// TwinCAT 3 PLC project Supervisorio
// ProgramVersion: 3.1.4024.0
// libraries:
//   CmpBitmapPool, * (System)
//   Tc2_Database, * (Beckhoff Automation GmbH)
//   Tc2_Standard, * (Beckhoff Automation GmbH)
//   Tc2_System, * (Beckhoff Automation GmbH)
//   Tc2_Utilities, * (Beckhoff Automation GmbH)
//   Tc3_EventLogger, * (Beckhoff Automation GmbH)
//   Tc3_Module, * (Beckhoff Automation GmbH)
//   VisuDialogs, * (System)
//   VisuSymbols,3.5.10.0,System
// project tree:
//   DUTs/ paPositions.TcDUT, raPositions.TcDUT, selectHist.TcDUT, statusEstufa.TcDUT, st_csv.TcDUT, tempData.TcDUT, timeDry.TcDUT (not stored)
//   / GlobalTextList.TcGTLO, PlcTask.TcTTO (not stored), Visualization Manager.TcVMO (not stored), VISU_TASK.TcTTO
//   GVLs/ GVL.TcGVL, GVL_C.TcGVL, GVL_P.TcGVL
//   POUs/Botons/ confirmSetInicio.TcPOU, confirmSecagem.TcPOU, gravarConfigPosicao.TcPOU, gravarConfigPosicao020.TcPOU, gravarConfigPosicao021.TcPOU, gravarConfigPosicao_Reator.TcPOU, gravarConfigPosicao_Reator_3.TcPOU, gravarConfigPosicao_Reator_2.TcPOU, iniciaProgramacaoEstufa.TcPOU, posCarrinho.TcPOU, posCarrinho2.TcPOU (not stored), posCarrinho3.TcPOU, selectPos021.TcPOU (not stored), selectPos019.TcPOU (not stored), selectPos020.TcPOU (not stored), simIniciaProg.TcPOU (not stored), simIniciaProg_Manual.TcPOU, simIniciaProg_Manual_3.TcPOU, simIniciaProg_Manual_2.TcPOU
//   POUs/ Chart_Gen.TcPOU, historical.TcPOU, MAIN.TcPOU, POU_Persistent.TcPOU, P_TextModeWrite.TcPOU, registerProc.TcPOU, registerProc20.TcPOU, registerProc21.TcPOU, registradorLog.TcPOU, registradorLog20.TcPOU, registradorLog21.TcPOU, ReportGenerator.TcPOU, Rotina019.TcPOU, Rotina019_Manual.TcPOU, Rotina021_Manual.TcPOU, Rotina020.TcPOU, Rotina021.TcPOU, Rotina020_Manual.TcPOU
//   VISUs/ Aba_Estufa.TcVIS, Aba_Estufa_2.TcVIS, Aba_Estufa_3.TcVIS (not stored), Aba_Manu.TcVIS, addComment.TcVIS, Carrinho_3.TcVIS (not stored), Carrinho_2.TcVIS (not stored), ConfigPosicao_3.TcVIS, ConfigPosicao_2.TcVIS, ConfigPosicao_Reator.TcVIS, ConfigPosicao_Reator_3.TcVIS (not stored), ConfigPosicao_Reator_2.TcVIS, Estufa2.TcVIS, Estufa3.TcVIS, FinalizaProg.TcVIS, Grafico_3.TcVIS, Grafico_2.TcVIS, Historical.TcVIS, IniciaProg_3.TcVIS, IniciaProg_2.TcVIS, Manu021.TcVIS, Manu020.TcVIS, Notifica24horas.TcVIS, Manu019.TcVIS, Carrinho.TcVIS, Estufa1.TcVIS, Grafico.TcVIS, Home.TcVIS, ImagePool.TcIPO (not stored), ConfigPosicao.TcVIS, IniciaProg.TcVIS (not stored), setInicio.TcVIS, setSecagem.TcVIS, TimeCustom.TcVIS, TimeCustom_3.TcVIS, TimeCustom_2.TcVIS
// real-time tasks:
//   TASK PlcTask: cycle T#10ms, priority 20, ADS port 350
//   TASK VISU_TASK: cycle T#200000us, priority 30, ADS port 351
// I/O:
//   DEVICE Device 1 (EtherCAT), AmsNetId 5.148.119.239.2.1
//     Term 1 (EK1200) [EK1200-5000 EtherCAT Power supply (2A E-Bus)]
//       Term 2 (EL6070) [EL6070 1Ch. Licensing-Terminal]
//       Term 3 (EL3058) [EL3058 8Ch. Ana. Input 4-20mA]
//       Term 4 (EL3052) [EL3052 2Ch. Ana. Input 4-20mA]
//       Term 5 (EL4008) [EL4008 8Ch. Ana. Output 0-10V, 12bit]
//       Term 6 (EL4002) [EL4002 2Ch. Ana. Output 0-10V, 12bit]
//       Term 7 (EL1809) [EL1809 16Ch. Dig. Input 24V, 3ms]
//       Term 8 (EL1809) [EL1809 16Ch. Dig. Input 24V, 3ms]
//       Term 9 (EL1809) [EL1809 16Ch. Dig. Input 24V, 3ms]
//       Term 10 (EL2809) [EL2809 16Ch. Dig. Output 24V, 0.5A]
//       Term 11 (EL2809) [EL2809 16Ch. Dig. Output 24V, 0.5A]
//       Term 12 (EL9011) [EL9011 End Terminal]
//   DEVICE Device 3 (NOV-DP-RAM)
// variable links:
//   Supervisorio/Supervisorio Instance <-> Device 1 (EtherCAT)/Term 1 (EK1200)/Term 10 (EL2809)
//     PlcTask Outputs/GVL.DigitalOut1[{1..16}] <-> Channel {1..16}/Output  (16 links)
//   Supervisorio/Supervisorio Instance <-> Device 1 (EtherCAT)/Term 1 (EK1200)/Term 11 (EL2809)
//     PlcTask Outputs/GVL.DigitalOut2[{1..16}] <-> Channel {1..16}/Output  (16 links)
//   Supervisorio/Supervisorio Instance <-> Device 1 (EtherCAT)/Term 1 (EK1200)/Term 3 (EL3058)
//     PlcTask Inputs/GVL.AnalogIn_4_20[{0..7}] <-> AI Standard Channel {1..8}/Value  (8 links)
//   Supervisorio/Supervisorio Instance <-> Device 1 (EtherCAT)/Term 1 (EK1200)/Term 4 (EL3052)
//     PlcTask Inputs/GVL.AnalogIn_4_20[8] <-> AI Standard Channel 1/Value
//     PlcTask Inputs/GVL.AnalogIn_4_20[9] <-> AI Standard Channel 2/Value
//   Supervisorio/Supervisorio Instance <-> Device 1 (EtherCAT)/Term 1 (EK1200)/Term 5 (EL4008)
//     PlcTask Outputs/GVL.AnalogOut_0_10[{0..7}] <-> AO Outputs Channel {1..8}/Analog output  (8 links)
//   Supervisorio/Supervisorio Instance <-> Device 1 (EtherCAT)/Term 1 (EK1200)/Term 6 (EL4002)
//     PlcTask Outputs/GVL.AnalogOut_0_10[8] <-> AO Outputs Channel 1/Analog output
//     PlcTask Outputs/GVL.AnalogOut_0_10[9] <-> AO Outputs Channel 2/Analog output
//   Supervisorio/Supervisorio Instance <-> Device 1 (EtherCAT)/Term 1 (EK1200)/Term 7 (EL1809)
//     PlcTask Inputs/GVL.DigitalIn1[{1..16}] <-> Channel {1..16}/Input  (16 links)
//   Supervisorio/Supervisorio Instance <-> Device 1 (EtherCAT)/Term 1 (EK1200)/Term 8 (EL1809)
//     PlcTask Inputs/GVL.DigitalIn2[{1..16}] <-> Channel {1..16}/Input  (16 links)
//   Supervisorio/Supervisorio Instance <-> Device 1 (EtherCAT)/Term 1 (EK1200)/Term 9 (EL1809)
//     PlcTask Inputs/GVL.DigitalIn3[{1..16}] <-> Channel {1..16}/Input  (16 links)

CONFIGURATION Supervisorio
    RESOURCE PLC ON TwinCAT3
        TASK VISU_TASK(INTERVAL := T#200000us, PRIORITY := 30);
        PROGRAM VisuElems_Visu_Prg WITH VISU_TASK : VisuElems.Visu_Prg;
    END_RESOURCE
END_CONFIGURATION

// ---- DUTs/paPositions.TcDUT
TYPE paPositions :
STRUCT
	cor: INT;
	color: DWORD;
	numOF: STRING;
	lote: STRING;
	text: string;
	class: REAL;
	pot: REAL;
	FP: INT;
	isolamento: int;
	reator: BOOL:= TRUE;
END_STRUCT
END_TYPE

// ---- DUTs/raPositions.TcDUT
TYPE raPositions :
STRUCT
	cor: INT;
	color: DWORD;
END_STRUCT
END_TYPE

// ---- DUTs/selectHist.TcDUT
TYPE selectHist :
STRUCT
	data: STRING(10);
	hora: STRING(10);
	auto: STRING(10);
	pos:  STRING(10);
	orfb: STRING(10);
	lote: STRING(10);
	class: STRING(50);
	pot: LREAL(8);
	isola: LREAL(8);
	fPot: STRING(10);
	reator: STRING(10);
	tempo: STRING(10);
	temp: DINT;
END_STRUCT
END_TYPE

// ---- DUTs/statusEstufa.TcDUT
TYPE statusEstufa :
STRUCT
	tempoSecagem: TIME; //DEFINIDO NA TELA ConfigPosicao
	tempoArmazenagem: TIME; //DEFINIDO NA TELA ConfigPosicao
	inicioSecagem: DATE_AND_TIME;
	fimSecagem: DATE_AND_TIME;
	prevFimSeca: DATE_AND_TIME;
	fimArmazenagem: DATE_AND_TIME;
	statusInicioSecagem: STRING;
	statusFimSecagem: STRING;
	statusFimArmazenagem: STRING;
	anoSec: STRING;
	mesSec: STRING;
	diaSec: STRING;
	horaSec: STRING;
	minutoSec: STRING;
	anoArm: STRING;
	mesArm: STRING;
	diaArm: STRING;
	horaArm: STRING;
	minutoArm: STRING;
	inicioReator: STRING;
	dtInicioReator: DATE_AND_TIME;
	start: BOOL;
	startManual: BOOL;
	tempSeca: INT;
	tempArm: int;
END_STRUCT
END_TYPE

// ---- DUTs/st_csv.TcDUT
TYPE st_csv :
STRUCT
	dia: STRING;
	mes: STRING;
	ano: STRING;
	ordem: STRING;
	lote: string;
END_STRUCT
END_TYPE

// ---- DUTs/tempData.TcDUT
TYPE tempData : 
STRUCT
	temp: REAL;
END_STRUCT
END_TYPE

// ---- GVLs/GVL.TcGVL
{attribute 'qualified_only'}
VAR_GLOBAL
	
////// Layout Interativo ////////

	
	
	corPos: DWORD;
	
  (*Pos Com Reator 00C000
	Pos Sem Reator FFFF00
	Pos Livre FFFFFF*)
	n: INT;
	i: INT;
	
	cfgPos_OF019: STRING;
	cfgPos_OF020: STRING;
	cfgPos_OF021: STRING;
	cfgPos_LT019: STRING;
	cfgPos_LT020: STRING;
	cfgPos_LT021: STRING;
	cfgPos_Class019: REAL;
	cfgPos_Class020: REAL;
	cfgPos_Class021: REAL;
	cfgPos_Pot019: REAL;
	cfgPos_Pot020: REAL;
	cfgPos_Pot021: REAL;
	cfgPos_Reat019: BOOL;
	cfgPos_Reat020: BOOL;
	cfgPos_Reat021: BOOL;
	cfgPos_FP019: INT;
	cfgPos_FP020: INT;
	cfgPos_FP021: INT;
	cfgPos_Iso019: INT;
	cfgPos_Iso020: INT;
	cfgPos_Iso021: INT;
	
	
	
////// Status Programação ///////////	

	
	logRegister: ARRAY[0..2] OF STRING;
	logRegister19: STRING;
	logRegister20: STRING;
	logRegister21: STRING;
	addTextLog: STRING;
	totalPos: ARRAY[0..2] OF INT;
	totalSeca: ARRAY[0..2] OF STRING;
	totalArm: ARRAY[0..2] OF STRING;
	totalRaet: ARRAY[0..2] OF INT;
	totalManual: ARRAY[0..2] OF INT;
	
	progInicio: ARRAY[0..2] OF STRING; //'DT#2024-3-31-23:59:0'
	progInicioReat: STRING;
	ano: STRING;
	mes: STRING;
	dia: STRING;
	hora: STRING;
	minuto: STRING;
	
	horaSecagem: STRING;
	minSecagem: STRING;
	horaArmazem: STRING;
	minArmazem: STRING;
	
	
	
	endSeca19: TIME;
	endSeca20: TIME;
	endSeca21: TIME;
	
	endArm19: TIME;
	endArm20: TIME;
	endArm21: TIME;
	
	
	
////// System Time ///////////	
	
	fbGetLocalSystemTime: FB_LocalSystemTime;
	sSystemDateTime: STRING;
	sSystemTime: STRING;
	sSystemDate: STRING;
	sDateTime: STRING;
	
	somaTempo: DATE_AND_TIME;
	
////// NÃO DEFINIDAS //////	
	actPos: INT;
	actEst: INT;
	actReat: INT;
	estAtiva: STRING;
	
	logButton: bool;
	
	bVentOn: BOOL;
	bAquecOn: BOOL;
	
	envialog: string;
	
	bstartchart019: BOOL;
	bstartchart020: BOOL;
	bstartchart021: BOOL;
	bAgendaInicio: BOOL;
	emergency: bool;
	
////// DECLARAÇÃO IOs //////

	AnalogIn_4_20 AT %I* : ARRAY[0..9] OF INT;
	AnalogOut_0_10 AT %Q* : ARRAY[0..9] OF INT;
	DigitalIn1 AT %I* : ARRAY[1..16] OF BOOL;
	DigitalIn2 AT %I* : ARRAY[1..16] OF BOOL;
	DigitalIn3 AT %I* : ARRAY[1..16] OF BOOL;
	DigitalOut1 AT %Q* : ARRAY[1..16] OF BOOL;
	DigitalOut2 AT %Q* : ARRAY[1..16] OF BOOL;
	
	
////// VARIAVEIS ESTUFA 019 //////

	zona1atual_019: REAL;
	zona2atual_019: REAL;
	zonaSegAtual_019: REAL;
	
	
	sobrecarga_M1_vent_019: BOOL;
	sobrecarga_M2_vent_019: BOOL;
	sobrecarga_Purga_019: BOOL;
	falhaTempHigh_019: BOOL;
	queimador1_block_019: BOOL;
	queimador2_block_019: BOOL;
	ventilacao_Ligada_019: BOOL;
	aquecimento_Desligado_019: BOOL;
	aquecimento_Ligado_019: BOOL;
	fimCicloAquecimento_019: BOOL;
	purgandoCamara_019: BOOL;
	liga_ventilacao_019: BOOL;
	liga_aquecimento_019: BOOL;
	desl_aquecimento_019: BOOL;
	emergencia019: BOOL;
	inEmergencia019: BOOL;
	
////// VARIAVEIS ESTUFA 020 //////

	zona1atual_020: REAL;
	zona2atual_020: REAL;
	zonaSegAtual_020: REAL;
	
	
	sobrecarga_M1_vent_020: BOOL;
	sobrecarga_M2_vent_020: BOOL;
	sobrecarga_Purga_020: BOOL;
	falhaTempHigh_020: BOOL;
	queimador1_block_020: BOOL;
	queimador2_block_020: BOOL;
	ventilacao_Ligada_020: BOOL;
	aquecimento_Desligado_020: BOOL;
	aquecimento_Ligado_020: BOOL;
	fimCicloAquecimento_020: BOOL;
	purgandoCamara_020: BOOL;
	liga_ventilacao_020: BOOL;
	liga_aquecimento_020: BOOL;
	desl_aquecimento_020: BOOL;	
	emergencia020: BOOL;
	inEmergencia020: BOOL;
	
////// VARIAVEIS ESTUFA 021 //////

	zona1atual_021: REAL;
	zona2atual_021: REAL;
	zonaSegAtual_021: REAL;
	
	
	sobrecarga_M1_vent_021: BOOL;
	sobrecarga_M2_vent_021: BOOL;
	sobrecarga_Purga_021: BOOL;
	falhaTempHigh_021: BOOL;
	queimador1_block_021: BOOL;
	queimador2_block_021: BOOL;
	ventilacao_Ligada_021: BOOL;
	aquecimento_Desligado_021: BOOL;
	aquecimento_Ligado_021: BOOL;
	fimCicloAquecimento_021: BOOL;
	purgandoCamara_021: BOOL;
	liga_ventilacao_021: BOOL;
	liga_aquecimento_021: BOOL;
	desl_aquecimento_021: BOOL;	
	emergencia021: BOOL;
	inEmergencia021: BOOL;
	
////// VARIAVEIS PRODWIN /////

	pwProd_019: BOOL;
	pwProd_020: BOOL;
	pwProd_021: BOOL;
	pwEmerg_019: BOOL;
	pwEmerg_020: BOOL;
	pwEmerg_021: BOOL;
	
////// VARIAVEI SQL //////

	sCmdInsertLog: STRING(3000);//INSERT INTO [dbo].[LogGeneral] ([HistoricalTime],[Description])VALUES('historicaltime','Description')
	//SELECT * FROM [dbo].[LogGeneral]
	sCmdInsertProc: STRING(3000);//INSERT INTO [dbo].[ProcessTable] ([data],[hora],[estufa],[auto],[user],[codPeca],[OF],[lote],[class],[pot],[isola],[fPot],[reator],[TIME],[temp])
	//VALUES ('data', 'hora', estufa0, 'auto', 'user', 'codpeca', 'OF', 'lote',	class0,	pot0, isola0, Fp0.0, 'reator', 'tempo',	tempe0)

	sCmdSelect19: STRING(3000);//'SELECT [data],[hora],[auto],[pos],[OF],[lote],[class],[pot],[isola],[fPot],[reator],[time],[temp] FROM [dbo].[ProcessTable19] WHERE data=$'2024-10-24$';';
	sCmdSelect20: STRING(3000);
	sCmdSelect21: STRING(3000);
	
	bInsertLog: BOOL;
	bInsertProc: BOOL;
	bSelect19: BOOL;
	aSelect19: ARRAY[1..MAX_CSV_ROWS] OF selecthist;
	bSelect20: BOOL;
	aSelect20: ARRAY[1..MAX_CSV_ROWS] OF selecthist;
	bSelect21: BOOL;
	aSelect21: ARRAY[1..MAX_CSV_ROWS] OF selecthist;
	
	permanencia: ARRAY[1..3] OF TIME;
	sReator: STRING;
	sFp: STRING;
	sIso: STRING;
	sAuto: STRING;
	bHistory: bool;
	
////// VARIAVEIS CSV //////
	
	report19: BOOL;
	radioFiltro: INT;
	radioEstufa: INT;
	radioData: BOOL;
	radioOF: BOOL;
	radioLote: BOOL;
	arrCVSfilter: ARRAY[0..2] OF st_csv;
	
	database: ARRAY[0..MAX_CSV_ROWS, 0..MAX_CSV_COLUMNS] OF STRING(MAX_CSV_FIELD_LENGTH); (*[ (* Source PLC database *)
	'0_0', '0_1', '0_2', '0_3', '0_4', '0_5',
	'1', '1_1', '1_2', '1_3', '1_4', '1_5',
	'2_0', '2_1', '2_2', '2_3', '2_4', '2_5',
	'3_0', '3_1', '3_2', '3_3', '3_4', '3_5',
	'4_0', '4_1', '4_2', '4_3', '4_4', '4_5',
	'5_0', '5_1', '5_2', '5_3', '5_4', '5_5'];*)
	
END_VAR

// ---- GVLs/GVL_C.TcGVL
VAR_GLOBAL CONSTANT
	MAX_CSV_ROWS 			: UDINT := 10000;
	MAX_CSV_COLUMNS 		: UDINT := 14;
	MAX_CSV_FIELD_LENGTH	: UDINT := 50;
END_VAR

// ---- GVLs/GVL_P.TcGVL
{attribute 'qualified_only'}
VAR_GLOBAL PERSISTENT
	
////// VARIAVEIS ESTUFA 019 //////

	zona1setpt_019: INT;
	zona2setpt_019: INT;
	zonaSegSetpt_019: INT;
	setPoint_019: INT;
	arr_Iso_1: ARRAY[0..3] OF INT;
	arr_FP_1: ARRAY[0..3] OF STRING;
	arr_CustomTime: ARRAY[0..1,1..10] OF INT;
	
////// VARIAVEIS ESTUFA 020 //////

	zona1setpt_020: INT;
	zona2setpt_020: INT;
	zonaSegSetpt_020: INT;
	setPoint_020: INT;
	arr_Iso_2: ARRAY[0..3] OF INT;
	arr_FP_2: ARRAY[0..3] OF STRING;
	arr_CustomTime_020: ARRAY[0..1,1..10] OF INT;
	
////// VARIAVEIS ESTUFA 021 //////

	zona1setpt_021: INT;
	zona2setpt_021: INT;
	zonaSegSetpt_021: INT;
	setPoint_021: INT;	
	arr_Iso_3: ARRAY[0..3] OF INT;
	arr_FP_3: ARRAY[0..3] OF STRING;
	arr_CustomTime_021: ARRAY[0..1,1..10] OF INT;
	
////// STATUS PROGRAMAÇÃO /////

	arrStatusEstufas: ARRAY[0..2] OF statusEstufa;
	etapa_process: ARRAY[0..2] OF STRING;
	
	arrLogEstufa19: ARRAY[1..100] OF STRING;
	arrLogEstufa20: ARRAY[1..100] OF STRING;
	arrLogEstufa21: ARRAY[1..100] OF STRING;
	
	
////// GRAFICO /////////

	arrTemp019: ARRAY[1..720] OF REAL;
	arrTempVisu019: ARRAY[1..720] OF REAL;
	arrTemp020: ARRAY[1..720] OF REAL;
	arrTempVisu020: ARRAY[1..720] OF REAL;
	arrTemp021: ARRAY[1..720] OF REAL;
	arrTempVisu021: ARRAY[1..720] OF REAL;
	
///// LAYOUT INTERATIVO /////

 	aReatorE019: ARRAY[1..2, 1..3] OF INT;
	aPositionsE019: ARRAY[1..24] OF paPositions;
	aReatorE020: ARRAY[1..2, 1..3] OF INT;
	aPositionsE020: ARRAY[1..24] OF paPositions;
	aReatorE021: ARRAY[1..2, 1..3] OF INT;
	aPositionsE021: ARRAY[1..24] OF paPositions;
	
	bCarrinhoReator1: BOOL:= TRUE;
	bCarrinhoReator2: BOOL:= TRUE;
	bCarrinhoReator3: BOOL:= TRUE;
	
	corPosReator1: ARRAY[1..6] OF raPositions;
	corPosReator2: ARRAY[1..6] OF raPositions;
	corPosReator3: ARRAY[1..6] OF raPositions;
	
END_VAR

// ---- POUs/Botons/confirmSetInicio.TcPOU
PROGRAM confirmSetInicio
VAR
END_VAR

gvl.progInicio[gvl.actEst]:= 'DT#20';
gvl.progInicio[gvl.actEst]:= concat(gvl.progInicio[gvl.actEst],gvl.ano);
gvl.progInicio[gvl.actEst]:= concat(gvl.progInicio[gvl.actEst],'-');
gvl.progInicio[gvl.actEst]:= concat(gvl.progInicio[gvl.actEst],gvl.mes);
gvl.progInicio[gvl.actEst]:= concat(gvl.progInicio[gvl.actEst],'-');
gvl.progInicio[gvl.actEst]:= concat(gvl.progInicio[gvl.actEst],gvl.dia);
gvl.progInicio[gvl.actEst]:= concat(gvl.progInicio[gvl.actEst],'-');
gvl.progInicio[gvl.actEst]:= concat(gvl.progInicio[gvl.actEst],gvl.hora);
gvl.progInicio[gvl.actEst]:= concat(gvl.progInicio[gvl.actEst],':');
gvl.progInicio[gvl.actEst]:= concat(gvl.progInicio[gvl.actEst],gvl.minuto);
gvl.progInicio[gvl.actEst]:= concat(gvl.progInicio[gvl.actEst],':0');

END_PROGRAM

// ---- POUs/Botons/confirmSecagem.TcPOU
PROGRAM confirmSecagem
VAR
	tempSeca: STRING;
	
END_VAR

//ESTE PROGRAMA TRANSFORMA O INPUT DO DIALOG EM TEMPO DE SECAGEM

tempSeca:= 'T#';
tempSeca:= concat(tempseca, TIME_TO_STRING(gvl_p.arrStatusEstufas[2].tempoSecagem));
tempSeca:= concat(tempseca, 'H');

GVL_p.arrStatusEstufas[2].tempoSecagem := STRING_TO_TIME(tempSeca);

END_PROGRAM

// ---- POUs/Botons/gravarConfigPosicao.TcPOU
PROGRAM gravarConfigPosicao
VAR
	bReator: ARRAY[0..2] OF BOOL;
	posicaoAtual: STRING;
	enviaLog: STRING;
	estufaAtual: STRING;
END_VAR

// CONTABILIZA A POSIÇÃO TOTAL  MUST BE FIRST-----------------------------------------------------------------

IF gvl_p.aPositionsE019[gvl.actPos].cor = 0 THEN
	gvl.totalPos[0]:= gvl.totalPos[0]+1;			
END_IF

// VERIFICA SE HA REATOR E MUDA A COR DO QUADRADO ------------------------------------
IF bReator[0] THEN
	gvl_p.aPositionsE019[gvl.actPos].cor:= 1;
	//gvl_p.bCarrinhoReator1:=TRUE;
	gvl.cfgPos_Reat019:=TRUE;
	ELSE
		gvl_p.aPositionsE019[gvl.actPos].cor:=2;
		//gvl_p.bCarrinhoReator1:=FALSE;
		gvl.cfgPos_Reat019:=FALSE;
END_IF

// REGISTRA AS INFORMAÇÕES EM CADA POSIÇÃO -------------------------------------------------------------
FOR gvl.n:=1 TO 24 BY 1 DO
	IF gvl.actPos = gvl.n THEN
		gvl_p.aPositionsE019[gvl.n].numOF:= gvl.cfgPos_OF019;
		gvl_p.aPositionsE019[gvl.n].lote:= gvl.cfgPos_LT019;
		gvl_p.aPositionsE019[gvl.n].class:= gvl.cfgPos_Class019;
		gvl_p.aPositionsE019[gvl.n].pot:= gvl.cfgPos_Pot019;
		gvl_p.aPositionsE019[gvl.n].reator:= gvl.cfgPos_Reat019;
		gvl_p.aPositionsE019[gvl.n].FP:= gvl.cfgPos_FP019;
		gvl_p.aPositionsE019[gvl.n].isolamento:= gvl.cfgPos_Iso019;
		gvl_p.aPositionsE019[gvl.n].text:= insert(gvl.cfgPos_OF019,'-',5);
		gvl_p.aPositionsE019[gvl.n].text:= concat(gvl_p.aPositionsE019[gvl.n].text,gvl.cfgPos_LT019);
	END_IF
END_FOR

// DEFINIÇÃO DOS TEMPOS DE ACORDO COM AS CLASSES ----------------------------------------------
(*IF gvl_p.aPositionsE019[gvl.actPos].class <= 15 THEN
		GVL_p.arrStatusEstufas[gvl.actEst].tempoSecagem := T#60H;
		GVL_p.arrStatusEstufas[gvl.actEst].tempoArmazenagem := T#192H;
		gvl.totalSeca[0]:= '60';
		gvl_p.arrStatusEstufas[gvl.actEst].tempSeca:= 120;
		gvl.totalArm[0]:= '192';
		gvl_p.arrStatusEstufas[gvl.actEst].tempArm:= 70;
		ELSIF gvl_p.aPositionsE019[gvl.actPos].class > 15 THEN
			GVL_p.arrStatusEstufas[gvl.actEst].tempoSecagem:= T#96H;
			GVL_p.arrStatusEstufas[gvl.actEst].tempoArmazenagem:= T#240H;
			gvl.totalSeca[0]:= '96';
			gvl_p.arrStatusEstufas[gvl.actEst].tempSeca:= 120;
			gvl.totalArm[0]:= '240';
			gvl_p.arrStatusEstufas[gvl.actEst].tempArm:= 70;
END_IF*)
IF gvl_p.aPositionsE019[gvl.actPos].pot <= 750 AND gvl_p.aPositionsE019[gvl.actPos].isolamento <= 25 AND gvl_p.aPositionsE019[gvl.actPos].FP = 1 THEN
	GVL_p.arrStatusEstufas[0].tempoSecagem := T#60H;
	GVL_p.arrStatusEstufas[0].tempoArmazenagem := T#192H;
	gvl.totalSeca[0]:= '60';
	gvl_p.arrStatusEstufas[0].tempSeca:= 120;
	gvl.totalArm[0]:= '192';
	gvl_p.arrStatusEstufas[0].tempArm:= 70;
	ELSIF gvl_p.aPositionsE019[gvl.actPos].pot <= 750 AND gvl_p.aPositionsE019[gvl.actPos].isolamento > 25 AND gvl_p.aPositionsE019[gvl.actPos].FP = 1 THEN
		GVL_p.arrStatusEstufas[0].tempoSecagem:= T#96H;
		GVL_p.arrStatusEstufas[0].tempoArmazenagem:= T#240H;
		gvl.totalSeca[0]:= '96';
		gvl_p.arrStatusEstufas[0].tempSeca:= 120;
		gvl.totalArm[0]:= '240';
		gvl_p.arrStatusEstufas[0].tempArm:= 70;
	ELSIF gvl_p.aPositionsE019[gvl.actPos].pot > 750 AND gvl_p.aPositionsE019[gvl.actPos].FP = 1 THEN
		GVL_p.arrStatusEstufas[0].tempoSecagem:= T#96H;
		GVL_p.arrStatusEstufas[0].tempoArmazenagem:= T#240H;
		gvl.totalSeca[0]:= '96';
		gvl_p.arrStatusEstufas[0].tempSeca:= 120;
		gvl.totalArm[0]:= '240';
		gvl_p.arrStatusEstufas[0].tempArm:= 70;
	ELSIF gvl_p.aPositionsE019[gvl.actPos].pot <= 750 AND gvl_p.aPositionsE019[gvl.actPos].isolamento <= 25 AND gvl_p.aPositionsE019[gvl.actPos].FP = 2 THEN
		GVL_p.arrStatusEstufas[0].tempoSecagem:= T#72H;
		GVL_p.arrStatusEstufas[0].tempoArmazenagem:= T#240H;
		gvl.totalSeca[0]:= '72';
		gvl_p.arrStatusEstufas[0].tempSeca:= 120;
		gvl.totalArm[0]:= '240';
		gvl_p.arrStatusEstufas[0].tempArm:= 70;
	ELSIF gvl_p.aPositionsE019[gvl.actPos].pot <= 750 AND gvl_p.aPositionsE019[gvl.actPos].isolamento > 25 AND gvl_p.aPositionsE019[gvl.actPos].FP = 2 THEN
		GVL_p.arrStatusEstufas[0].tempoSecagem:= T#96H;
		GVL_p.arrStatusEstufas[0].tempoArmazenagem:= T#240H;
		gvl.totalSeca[0]:= '96';
		gvl_p.arrStatusEstufas[0].tempSeca:= 120;
		gvl.totalArm[0]:= '240';
		gvl_p.arrStatusEstufas[0].tempArm:= 70;
	ELSIF gvl_p.aPositionsE019[gvl.actPos].pot > 750 AND gvl_p.aPositionsE019[gvl.actPos].FP = 2 THEN
		GVL_p.arrStatusEstufas[0].tempoSecagem:= T#96H;
		GVL_p.arrStatusEstufas[0].tempoArmazenagem:= T#240H;
		gvl.totalSeca[0]:= '96';
		gvl_p.arrStatusEstufas[0].tempSeca:= 120;
		gvl.totalArm[0]:= '240';
		gvl_p.arrStatusEstufas[0].tempArm:= 70;	
END_IF

///// GERADOR DE LOG -------------------------------------------------------------

posicaoAtual:= INT_TO_STRING(gvl.actPos);
estufaAtual:= INT_TO_STRING(gvl.actEst);
envialog:= 'Posição Nº ';
enviaLog:= concat(envialog, posicaoAtual);
enviaLog:= concat(envialog,' gravada. ESTUFA 019');
gvl.logRegister19:= envialog;

gvl.sCmdInsertLog:= 'INSERT INTO [dbo].[LogGeneral] ([HistoricalTime],[Description])VALUES($'$',$'$')';
gvl.sCmdInsertLog:= insert(gvl.sCmdInsertLog,gvl.logRegister19,74);	
gvl.sCmdInsertLog:= insert(gvl.sCmdInsertLog,gvl.sSystemDateTime,71);
gvl.bInsertLog:= TRUE;

END_PROGRAM

// ---- POUs/Botons/gravarConfigPosicao020.TcPOU
PROGRAM gravarConfigPosicao020
VAR
	bReator: ARRAY[0..2] OF BOOL;
	posicaoAtual: STRING;
	enviaLog: STRING;
	estufaAtual: STRING;
END_VAR

// CONTABILIZA A POSIÇÃO TOTAL  MUST BE FIRST-----------------------------------------------------------------

IF gvl_p.aPositionsE020[gvl.actPos].cor = 0 THEN
	gvl.totalPos[1]:= gvl.totalPos[1]+1;			
END_IF

// VERIFICA SE HA REATOR E MUDA A COR DO QUADRADO ------------------------------------
IF bReator[1] THEN
	gvl_p.aPositionsE020[gvl.actPos].cor:= 1;
	//gvl_p.bCarrinhoReator2:=TRUE;
	gvl.cfgPos_Reat020:=TRUE;
	ELSE
		gvl_p.aPositionsE020[gvl.actPos].cor:=2;
		//gvl_p.bCarrinhoReator2:=FALSE;
		gvl.cfgPos_Reat020:=FALSE;
END_IF

// REGISTRA AS INFORMAÇÕES EM CADA POSIÇÃO -------------------------------------------------------------
FOR gvl.n:=1 TO 24 BY 1 DO
	IF gvl.actPos = gvl.n THEN
		gvl_p.aPositionsE020[gvl.n].numOF:= gvl.cfgPos_OF020;
		gvl_p.aPositionsE020[gvl.n].lote:= gvl.cfgPos_LT020;
		gvl_p.aPositionsE020[gvl.n].class:= gvl.cfgPos_Class020;
		gvl_p.aPositionsE020[gvl.n].pot:= gvl.cfgPos_Pot020;
		gvl_p.aPositionsE020[gvl.n].reator:= gvl.cfgPos_Reat020;
		gvl_p.aPositionsE020[gvl.n].FP:= gvl.cfgPos_FP020;
		gvl_p.aPositionsE020[gvl.n].isolamento:= gvl.cfgPos_Iso020;
		gvl_p.aPositionsE020[gvl.n].text:= insert(gvl.cfgPos_OF020,'-',5);
		gvl_p.aPositionsE020[gvl.n].text:= concat(gvl_p.aPositionsE020[gvl.n].text,gvl.cfgPos_LT020);
	END_IF
END_FOR

// DEFINIÇÃO DOS TEMPOS DE ACORDO COM AS CLASSES ----------------------------------------------
(*IF gvl_p.aPositionsE020[gvl.actPos].class <= 15 THEN
		GVL_p.arrStatusEstufas[gvl.actEst].tempoSecagem := T#60H;
		GVL_p.arrStatusEstufas[gvl.actEst].tempoArmazenagem := T#192H;
		gvl.totalSeca[1]:= '60';
		gvl_p.arrStatusEstufas[gvl.actEst].tempSeca:= 120;
		gvl.totalArm[1]:= '192';
		gvl_p.arrStatusEstufas[gvl.actEst].tempArm:= 70;
		ELSIF gvl_p.aPositionsE020[gvl.actPos].class > 15 THEN
			GVL_p.arrStatusEstufas[gvl.actEst].tempoSecagem:= T#96H;
			GVL_p.arrStatusEstufas[gvl.actEst].tempoArmazenagem:= T#240H;
			gvl.totalSeca[1]:= '96';
			gvl_p.arrStatusEstufas[gvl.actEst].tempSeca:= 120;
			gvl.totalArm[1]:= '240';
			gvl_p.arrStatusEstufas[gvl.actEst].tempArm:= 70;
END_IF*)
IF gvl_p.aPositionsE020[gvl.actPos].pot <= 750 AND gvl_p.aPositionsE020[gvl.actPos].isolamento <= 25 AND gvl_p.aPositionsE020[gvl.actPos].FP = 1 THEN
	GVL_p.arrStatusEstufas[1].tempoSecagem := T#60H;
	GVL_p.arrStatusEstufas[1].tempoArmazenagem := T#192H;
	gvl.totalSeca[1]:= '60';
	gvl_p.arrStatusEstufas[1].tempSeca:= 120;
	gvl.totalArm[1]:= '192';
	gvl_p.arrStatusEstufas[1].tempArm:= 70;
	ELSIF gvl_p.aPositionsE020[gvl.actPos].pot <= 750 AND gvl_p.aPositionsE020[gvl.actPos].isolamento > 25 AND gvl_p.aPositionsE020[gvl.actPos].FP = 1 THEN
		GVL_p.arrStatusEstufas[1].tempoSecagem:= T#96H;
		GVL_p.arrStatusEstufas[1].tempoArmazenagem:= T#240H;
		gvl.totalSeca[1]:= '96';
		gvl_p.arrStatusEstufas[1].tempSeca:= 120;
		gvl.totalArm[1]:= '240';
		gvl_p.arrStatusEstufas[1].tempArm:= 70;
	ELSIF gvl_p.aPositionsE020[gvl.actPos].pot > 750 AND gvl_p.aPositionsE020[gvl.actPos].FP = 1 THEN
		GVL_p.arrStatusEstufas[1].tempoSecagem:= T#96H;
		GVL_p.arrStatusEstufas[1].tempoArmazenagem:= T#240H;
		gvl.totalSeca[1]:= '96';
		gvl_p.arrStatusEstufas[1].tempSeca:= 120;
		gvl.totalArm[1]:= '240';
		gvl_p.arrStatusEstufas[1].tempArm:= 70;
	ELSIF gvl_p.aPositionsE020[gvl.actPos].pot <= 750 AND gvl_p.aPositionsE020[gvl.actPos].isolamento <= 25 AND gvl_p.aPositionsE020[gvl.actPos].FP = 2 THEN
		GVL_p.arrStatusEstufas[1].tempoSecagem:= T#72H;
		GVL_p.arrStatusEstufas[1].tempoArmazenagem:= T#240H;
		gvl.totalSeca[1]:= '72';
		gvl_p.arrStatusEstufas[1].tempSeca:= 120;
		gvl.totalArm[1]:= '240';
		gvl_p.arrStatusEstufas[1].tempArm:= 70;
	ELSIF gvl_p.aPositionsE020[gvl.actPos].pot <= 750 AND gvl_p.aPositionsE020[gvl.actPos].isolamento > 25 AND gvl_p.aPositionsE020[gvl.actPos].FP = 2 THEN
		GVL_p.arrStatusEstufas[1].tempoSecagem:= T#96H;
		GVL_p.arrStatusEstufas[1].tempoArmazenagem:= T#240H;
		gvl.totalSeca[1]:= '96';
		gvl_p.arrStatusEstufas[1].tempSeca:= 120;
		gvl.totalArm[1]:= '240';
		gvl_p.arrStatusEstufas[1].tempArm:= 70;
	ELSIF gvl_p.aPositionsE020[gvl.actPos].pot > 750 AND gvl_p.aPositionsE020[gvl.actPos].FP = 2 THEN
		GVL_p.arrStatusEstufas[1].tempoSecagem:= T#96H;
		GVL_p.arrStatusEstufas[1].tempoArmazenagem:= T#240H;
		gvl.totalSeca[1]:= '96';
		gvl_p.arrStatusEstufas[1].tempSeca:= 120;
		gvl.totalArm[1]:= '240';
		gvl_p.arrStatusEstufas[1].tempArm:= 70;	
END_IF

///// GERADOR DE LOG -------------------------------------------------------------

posicaoAtual:= INT_TO_STRING(gvl.actPos);
estufaAtual:= INT_TO_STRING(gvl.actEst);
envialog:= 'Posição Nº ';
enviaLog:= concat(envialog, posicaoAtual);
enviaLog:= concat(envialog,' gravada.  ESTUFA 020');
gvl.logRegister20:= envialog;

gvl.sCmdInsertLog:= 'INSERT INTO [dbo].[LogGeneral] ([HistoricalTime],[Description])VALUES($'$',$'$')';
gvl.sCmdInsertLog:= insert(gvl.sCmdInsertLog,gvl.logRegister20,74);	
gvl.sCmdInsertLog:= insert(gvl.sCmdInsertLog,gvl.sSystemDateTime,71);
gvl.bInsertLog:= TRUE;

END_PROGRAM

// ---- POUs/Botons/gravarConfigPosicao021.TcPOU
PROGRAM gravarConfigPosicao021
VAR
	bReator: ARRAY[0..2] OF BOOL;
	posicaoAtual: STRING;
	enviaLog: STRING;
	estufaAtual: STRING;
END_VAR

// CONTABILIZA A POSIÇÃO TOTAL  MUST BE FIRST-----------------------------------------------------------------

IF gvl_p.aPositionsE021[gvl.actPos].cor = 0 THEN
		gvl.totalPos[2]:= gvl.totalPos[2]+1;			
	END_IF
	
// VERIFICA SE HA REATOR E MUDA A COR DO QUADRADO ------------------------------------
IF bReator[2] THEN
	gvl_p.aPositionsE021[gvl.actPos].cor:= 1;
	//gvl_p.bCarrinhoReator3:=TRUE;
	gvl.cfgPos_Reat021:=TRUE;
	ELSE
		gvl_p.aPositionsE021[gvl.actPos].cor:=2;
		//gvl_p.bCarrinhoReator3:=FALSE;
		gvl.cfgPos_Reat021:=FALSE;	
END_IF

// REGISTRA AS INFORMAÇÕES EM CADA POSIÇÃO -------------------------------------------------------------
FOR gvl.n:=1 TO 24 BY 1 DO
	IF gvl.actPos = gvl.n THEN
		gvl_p.aPositionsE021[gvl.n].numOF:= gvl.cfgPos_OF021;
		gvl_p.aPositionsE021[gvl.n].lote:= gvl.cfgPos_LT021;
		gvl_p.aPositionsE021[gvl.n].class:= gvl.cfgPos_Class021;
		gvl_p.aPositionsE021[gvl.n].pot:= gvl.cfgPos_Pot021;
		gvl_p.aPositionsE021[gvl.n].reator:= gvl.cfgPos_Reat021;
		gvl_p.aPositionsE021[gvl.n].FP:= gvl.cfgPos_FP021;
		gvl_p.aPositionsE021[gvl.n].isolamento:= gvl.cfgPos_Iso021;
		gvl_p.aPositionsE021[gvl.n].text:= insert(gvl.cfgPos_OF021,'-',5);
		gvl_p.aPositionsE021[gvl.n].text:= concat(gvl_p.aPositionsE021[gvl.n].text,gvl.cfgPos_LT021);
	END_IF
END_FOR

// DEFINIÇÃO DOS TEMPOS DE ACORDO COM AS CLASSES ----------------------------------------------
(*IF gvl_p.aPositionsE021[gvl.actPos].class <= 15 THEN
		GVL_p.arrStatusEstufas[2].tempoSecagem := T#60H;
		GVL_p.arrStatusEstufas[2].tempoArmazenagem := T#192H;
		gvl.totalSeca[2]:= '60';
		gvl_p.arrStatusEstufas[2].tempSeca:= 120;
		gvl.totalArm[2]:= '192';
		gvl_p.arrStatusEstufas[2].tempArm:= 70;
		ELSIF gvl_p.aPositionsE021[gvl.actPos].class > 15 THEN
			GVL_p.arrStatusEstufas[2].tempoSecagem:= T#96H;
			GVL_p.arrStatusEstufas[2].tempoArmazenagem:= T#240H;
			gvl.totalSeca[2]:= '96';
			gvl_p.arrStatusEstufas[2].tempSeca:= 120;
			gvl.totalArm[2]:= '240';
			gvl_p.arrStatusEstufas[2].tempArm:= 70;
END_IF*)
IF gvl_p.aPositionsE021[gvl.actPos].pot <= 750 AND gvl_p.aPositionsE021[gvl.actPos].isolamento <= 25 AND gvl_p.aPositionsE021[gvl.actPos].FP = 1 THEN
	GVL_p.arrStatusEstufas[2].tempoSecagem := T#60H;
	GVL_p.arrStatusEstufas[2].tempoArmazenagem := T#192H;
	gvl.totalSeca[2]:= '60';
	gvl_p.arrStatusEstufas[2].tempSeca:= 120;
	gvl.totalArm[2]:= '192';
	gvl_p.arrStatusEstufas[2].tempArm:= 70;
	ELSIF gvl_p.aPositionsE021[gvl.actPos].pot <= 750 AND gvl_p.aPositionsE021[gvl.actPos].isolamento > 25 AND gvl_p.aPositionsE021[gvl.actPos].FP = 1 THEN
		GVL_p.arrStatusEstufas[2].tempoSecagem:= T#96H;
		GVL_p.arrStatusEstufas[2].tempoArmazenagem:= T#240H;
		gvl.totalSeca[2]:= '96';
		gvl_p.arrStatusEstufas[2].tempSeca:= 120;
		gvl.totalArm[2]:= '240';
		gvl_p.arrStatusEstufas[2].tempArm:= 70;
	ELSIF gvl_p.aPositionsE021[gvl.actPos].pot > 750 AND gvl_p.aPositionsE021[gvl.actPos].FP = 1 THEN
		GVL_p.arrStatusEstufas[2].tempoSecagem:= T#96H;
		GVL_p.arrStatusEstufas[2].tempoArmazenagem:= T#240H;
		gvl.totalSeca[2]:= '96';
		gvl_p.arrStatusEstufas[2].tempSeca:= 120;
		gvl.totalArm[2]:= '240';
		gvl_p.arrStatusEstufas[2].tempArm:= 70;
	ELSIF gvl_p.aPositionsE021[gvl.actPos].pot <= 750 AND gvl_p.aPositionsE021[gvl.actPos].isolamento <= 25 AND gvl_p.aPositionsE021[gvl.actPos].FP = 2 THEN
		GVL_p.arrStatusEstufas[2].tempoSecagem:= T#72H;
		GVL_p.arrStatusEstufas[2].tempoArmazenagem:= T#240H;
		gvl.totalSeca[2]:= '72';
		gvl_p.arrStatusEstufas[2].tempSeca:= 120;
		gvl.totalArm[2]:= '240';
		gvl_p.arrStatusEstufas[2].tempArm:= 70;
	ELSIF gvl_p.aPositionsE021[gvl.actPos].pot <= 750 AND gvl_p.aPositionsE021[gvl.actPos].isolamento > 25 AND gvl_p.aPositionsE021[gvl.actPos].FP = 2 THEN
		GVL_p.arrStatusEstufas[2].tempoSecagem:= T#96H;
		GVL_p.arrStatusEstufas[2].tempoArmazenagem:= T#240H;
		gvl.totalSeca[2]:= '96';
		gvl_p.arrStatusEstufas[2].tempSeca:= 120;
		gvl.totalArm[2]:= '240';
		gvl_p.arrStatusEstufas[2].tempArm:= 70;
	ELSIF gvl_p.aPositionsE021[gvl.actPos].pot > 750 AND gvl_p.aPositionsE021[gvl.actPos].FP = 2 THEN
		GVL_p.arrStatusEstufas[2].tempoSecagem:= T#96H;
		GVL_p.arrStatusEstufas[2].tempoArmazenagem:= T#240H;
		gvl.totalSeca[2]:= '96';
		gvl_p.arrStatusEstufas[2].tempSeca:= 120;
		gvl.totalArm[2]:= '240';
		gvl_p.arrStatusEstufas[2].tempArm:= 70;	
END_IF

///// GERADOR DE LOG -------------------------------------------------------------

posicaoAtual:= INT_TO_STRING(gvl.actPos);
estufaAtual:= INT_TO_STRING(gvl.actEst);
envialog:= 'Posição Nº ';
enviaLog:= concat(envialog, posicaoAtual);
enviaLog:= concat(envialog,' gravada.  ESTUFA 021');
gvl.logRegister21:= envialog;

gvl.sCmdInsertLog:= 'INSERT INTO [dbo].[LogGeneral] ([HistoricalTime],[Description])VALUES($'$',$'$')';
gvl.sCmdInsertLog:= insert(gvl.sCmdInsertLog,gvl.logRegister21,74);	
gvl.sCmdInsertLog:= insert(gvl.sCmdInsertLog,gvl.sSystemDateTime,71);
gvl.bInsertLog:= TRUE;

END_PROGRAM

// ---- POUs/Botons/gravarConfigPosicao_Reator.TcPOU
PROGRAM gravarConfigPosicao_Reator
VAR
	bReator: BOOL;
	posicaoAtual: STRING;
	enviaLog: STRING;
	somaReator: TIME;
	timeCalc: TIME;
	
	dia: STRING;
	mes: STRING;
	ano: STRING;
	hora: STRING;
	minuto: STRING;
	
	bGravarConfigPosicao_Reator: BOOL:= FALSE;
	
	bNotificaTime: BOOL;
	estufaAtual: STRING;
END_VAR


IF gvl.actEst = 0 THEN
gvl_p.corPosReator1[gvl.actReat].cor:= 1;
ELSIF gvl.actEst = 1 THEN
	gvl_p.corPosReator2[gvl.actReat].cor:= 1;
	ELSIF gvl.actEst = 2 THEN
		gvl_p.corPosReator3[gvl.actReat].cor:= 1;
		END_IF
	

///// IMPRIMIR A HORA E A DATA DO INICIO DA SECAGEM-------------------------------

IF simIniciaProg.bSimIniciaProg THEN
gvl.progInicioReat:= DT_TO_STRING(gvl.somaTempo);
gvl_p.arrStatusEstufas[gvl.actEst].dtInicioReator:= gvl.somaTempo;
dia:= MID(STR:= gvl.progInicioReat , LEN:= 2, POS:=12);
mes:= MID(STR:= gvl.progInicioReat , LEN:= 2, POS:=9);
ano:= MID(STR:= gvl.progInicioReat , LEN:= 2, POS:=6);
hora:= MID(STR:= gvl.progInicioReat , LEN:= 2, POS:=15);
minuto:= MID(STR:= gvl.progInicioReat , LEN:= 2, POS:=18);

gvl_p.arrStatusEstufas[gvl.actEst].inicioReator := '';
gvl_p.arrStatusEstufas[gvl.actEst].inicioReator := concat(gvl_p.arrStatusEstufas[gvl.actEst].inicioReator,hora);
gvl_p.arrStatusEstufas[gvl.actEst].inicioReator := concat(gvl_p.arrStatusEstufas[gvl.actEst].inicioReator,':');
gvl_p.arrStatusEstufas[gvl.actEst].inicioReator := concat(gvl_p.arrStatusEstufas[gvl.actEst].inicioReator,minuto);
gvl_p.arrStatusEstufas[gvl.actEst].inicioReator := concat(gvl_p.arrStatusEstufas[gvl.actEst].inicioReator,' ');
gvl_p.arrStatusEstufas[gvl.actEst].inicioReator := concat(gvl_p.arrStatusEstufas[gvl.actEst].inicioReator,dia);
gvl_p.arrStatusEstufas[gvl.actEst].inicioReator := concat(gvl_p.arrStatusEstufas[gvl.actEst].inicioReator,'/');
gvl_p.arrStatusEstufas[gvl.actEst].inicioReator := concat(gvl_p.arrStatusEstufas[gvl.actEst].inicioReator,mes);
gvl_p.arrStatusEstufas[gvl.actEst].inicioReator := concat(gvl_p.arrStatusEstufas[gvl.actEst].inicioReator,'/');
gvl_p.arrStatusEstufas[gvl.actEst].inicioReator := concat(gvl_p.arrStatusEstufas[gvl.actEst].inicioReator,ano);

///// CALCULO DE DEFINIÇÃO SE O PROCESSO PASSA DAS 36 HORAS LIMITES ----------------------------------------
timeCalc:= (gvl_p.arrStatusEstufas[gvl.actEst].prevFimSeca - systemtime_to_dt(gvl.fbGetLocalSystemTime.systemTime));
IF timeCalc < T#24H THEN
	gvl_P.arrStatusEstufas[gvl.actEst].fimSecagem := gvl_p.arrStatusEstufas[gvl.actEst].dtInicioReator + T#24H;
END_IF

///// DECOMPOR A VARIAVEL FIM DA SECAGEM -----------------------------------------------------------------------------------------------
gvl_p.arrStatusEstufas[gvl.actEst].diaSec := MID(STR:= DT_TO_STRING(gvl_p.arrStatusEstufas[gvl.actEst].fimSecagem) , LEN:= 2, POS:=12);
gvl_p.arrStatusEstufas[gvl.actEst].mesSec := MID(STR:= DT_TO_STRING(gvl_p.arrStatusEstufas[gvl.actEst].fimSecagem), LEN:= 2, POS:=9);
gvl_p.arrStatusEstufas[gvl.actEst].anoSec := MID(STR:= DT_TO_STRING(gvl_p.arrStatusEstufas[gvl.actEst].fimSecagem), LEN:= 2, POS:=6);
gvl_p.arrStatusEstufas[gvl.actEst].horaSec := MID(STR:= DT_TO_STRING(gvl_p.arrStatusEstufas[gvl.actEst].fimSecagem), LEN:= 2, POS:=15);
gvl_p.arrStatusEstufas[gvl.actEst].minutoSec := MID(STR:= DT_TO_STRING(gvl_p.arrStatusEstufas[gvl.actEst].fimSecagem), LEN:= 2, POS:=18);

///// IMPRIMIR A HORA E A DATA DO FIM DA SECAGEM --------------------------------------------------------------------------------------------------------
gvl_p.arrStatusEstufas[gvl.actEst].statusFimSecagem := '';
gvl_p.arrStatusEstufas[gvl.actEst].statusFimSecagem := concat(gvl_p.arrStatusEstufas[gvl.actEst].statusFimSecagem,gvl_p.arrStatusEstufas[gvl.actEst].horaSec);
gvl_p.arrStatusEstufas[gvl.actEst].statusFimSecagem := concat(gvl_p.arrStatusEstufas[gvl.actEst].statusFimSecagem,':');
gvl_p.arrStatusEstufas[gvl.actEst].statusFimSecagem := concat(gvl_p.arrStatusEstufas[gvl.actEst].statusFimSecagem,gvl_p.arrStatusEstufas[gvl.actEst].minutoSec);
gvl_p.arrStatusEstufas[gvl.actEst].statusFimSecagem := concat(gvl_p.arrStatusEstufas[gvl.actEst].statusFimSecagem,' ');
gvl_p.arrStatusEstufas[gvl.actEst].statusFimSecagem := concat(gvl_p.arrStatusEstufas[gvl.actEst].statusFimSecagem,gvl_p.arrStatusEstufas[gvl.actEst].diaSec);
gvl_p.arrStatusEstufas[gvl.actEst].statusFimSecagem := concat(gvl_p.arrStatusEstufas[gvl.actEst].statusFimSecagem,'/');
gvl_p.arrStatusEstufas[gvl.actEst].statusFimSecagem := concat(gvl_p.arrStatusEstufas[gvl.actEst].statusFimSecagem,gvl_p.arrStatusEstufas[gvl.actEst].mesSec);
gvl_p.arrStatusEstufas[gvl.actEst].statusFimSecagem := concat(gvl_p.arrStatusEstufas[gvl.actEst].statusFimSecagem,'/');
gvl_p.arrStatusEstufas[gvl.actEst].statusFimSecagem := concat(gvl_p.arrStatusEstufas[gvl.actEst].statusFimSecagem,gvl_p.arrStatusEstufas[gvl.actEst].anoSec);

///// DECOMPOR A VARIAVEL FIM DA ARMAZENAGEM -------------------------------------------------------------------------------------------
gvl_p.arrStatusEstufas[gvl.actEst].diaArm := MID(STR:= DT_TO_STRING(gvl_p.arrStatusEstufas[gvl.actEst].fimArmazenagem) , LEN:= 2, POS:=12);
gvl_p.arrStatusEstufas[gvl.actEst].mesArm := MID(STR:= DT_TO_STRING(gvl_p.arrStatusEstufas[gvl.actEst].fimArmazenagem), LEN:= 2, POS:=9);
gvl_p.arrStatusEstufas[gvl.actEst].anoArm := MID(STR:= DT_TO_STRING(gvl_p.arrStatusEstufas[gvl.actEst].fimArmazenagem), LEN:= 2, POS:=6);
gvl_p.arrStatusEstufas[gvl.actEst].horaArm := MID(STR:= DT_TO_STRING(gvl_p.arrStatusEstufas[gvl.actEst].fimArmazenagem), LEN:= 2, POS:=15);
gvl_p.arrStatusEstufas[gvl.actEst].minutoArm := MID(STR:= DT_TO_STRING(gvl_p.arrStatusEstufas[gvl.actEst].fimArmazenagem), LEN:= 2, POS:=18);

///// IMPRIMIR A HORA E A DATA DO FIM DA ARMAZENAGEM -----------------------------------------------------------------------------------------------------------
gvl_p.arrStatusEstufas[gvl.actEst].statusFimArmazenagem := '';
gvl_p.arrStatusEstufas[gvl.actEst].statusFimArmazenagem := concat(gvl_p.arrStatusEstufas[gvl.actEst].statusFimArmazenagem,gvl_p.arrStatusEstufas[gvl.actEst].horaArm);
gvl_p.arrStatusEstufas[gvl.actEst].statusFimArmazenagem := concat(gvl_p.arrStatusEstufas[gvl.actEst].statusFimArmazenagem,':');
gvl_p.arrStatusEstufas[gvl.actEst].statusFimArmazenagem := concat(gvl_p.arrStatusEstufas[gvl.actEst].statusFimArmazenagem,gvl_p.arrStatusEstufas[gvl.actEst].minutoArm);
gvl_p.arrStatusEstufas[gvl.actEst].statusFimArmazenagem := concat(gvl_p.arrStatusEstufas[gvl.actEst].statusFimArmazenagem,' ');
gvl_p.arrStatusEstufas[gvl.actEst].statusFimArmazenagem := concat(gvl_p.arrStatusEstufas[gvl.actEst].statusFimArmazenagem,gvl_p.arrStatusEstufas[gvl.actEst].diaArm);
gvl_p.arrStatusEstufas[gvl.actEst].statusFimArmazenagem := concat(gvl_p.arrStatusEstufas[gvl.actEst].statusFimArmazenagem,'/');
gvl_p.arrStatusEstufas[gvl.actEst].statusFimArmazenagem := concat(gvl_p.arrStatusEstufas[gvl.actEst].statusFimArmazenagem,gvl_p.arrStatusEstufas[gvl.actEst].mesArm);
gvl_p.arrStatusEstufas[gvl.actEst].statusFimArmazenagem := concat(gvl_P.arrStatusEstufas[gvl.actEst].statusFimArmazenagem,'/');
gvl_p.arrStatusEstufas[gvl.actEst].statusFimArmazenagem := concat(gvl_P.arrStatusEstufas[gvl.actEst].statusFimArmazenagem,gvl_p.arrStatusEstufas[gvl.actEst].anoArm);

END_IF

///// GERADOR DE LOG -------------------------------------------------------------

posicaoAtual:= INT_TO_STRING(gvl.actReat);
estufaAtual:= INT_TO_STRING(gvl.actEst);
envialog:= 'Reator adicionado a posição de Nº ';
enviaLog:= concat(envialog, posicaoAtual);
enviaLog:= concat(envialog, '.');
enviaLog:= concat(envialog, ' ESTUFA ');
enviaLog:= concat(envialog, estufaAtual);
gvl.logRegister19:= envialog;

bGravarConfigPosicao_Reator:= TRUE;

END_PROGRAM

// ---- POUs/Botons/gravarConfigPosicao_Reator_3.TcPOU
PROGRAM gravarConfigPosicao_Reator_3
VAR
	bReator: BOOL;
	posicaoAtual: STRING;
	enviaLog: STRING;
	somaReator: TIME;
	timeCalc: TIME;
	
	dia: STRING;
	mes: STRING;
	ano: STRING;
	hora: STRING;
	minuto: STRING;
	
	bGravarConfigPosicao_Reator: BOOL:= FALSE;
	
	bNotificaTime: BOOL;
	estufaAtual: STRING;
END_VAR


IF gvl.actEst = 0 THEN
gvl_p.corPosReator1[gvl.actReat].cor:= 1;
ELSIF gvl.actEst = 1 THEN
	gvl_p.corPosReator2[gvl.actReat].cor:= 1;
	ELSIF gvl.actEst = 2 THEN
		gvl_p.corPosReator3[gvl.actReat].cor:= 1;
		END_IF
	

///// IMPRIMIR A HORA E A DATA DO INICIO DA SECAGEM-------------------------------

IF simIniciaProg.bSimIniciaProg THEN
gvl.progInicioReat:= DT_TO_STRING(gvl.somaTempo);
gvl_p.arrStatusEstufas[gvl.actEst].dtInicioReator:= gvl.somaTempo;
dia:= MID(STR:= gvl.progInicioReat , LEN:= 2, POS:=12);
mes:= MID(STR:= gvl.progInicioReat , LEN:= 2, POS:=9);
ano:= MID(STR:= gvl.progInicioReat , LEN:= 2, POS:=6);
hora:= MID(STR:= gvl.progInicioReat , LEN:= 2, POS:=15);
minuto:= MID(STR:= gvl.progInicioReat , LEN:= 2, POS:=18);

gvl_p.arrStatusEstufas[gvl.actEst].inicioReator := '';
gvl_p.arrStatusEstufas[gvl.actEst].inicioReator := concat(gvl_p.arrStatusEstufas[gvl.actEst].inicioReator,hora);
gvl_p.arrStatusEstufas[gvl.actEst].inicioReator := concat(gvl_p.arrStatusEstufas[gvl.actEst].inicioReator,':');
gvl_p.arrStatusEstufas[gvl.actEst].inicioReator := concat(gvl_p.arrStatusEstufas[gvl.actEst].inicioReator,minuto);
gvl_p.arrStatusEstufas[gvl.actEst].inicioReator := concat(gvl_p.arrStatusEstufas[gvl.actEst].inicioReator,' ');
gvl_p.arrStatusEstufas[gvl.actEst].inicioReator := concat(gvl_p.arrStatusEstufas[gvl.actEst].inicioReator,dia);
gvl_p.arrStatusEstufas[gvl.actEst].inicioReator := concat(gvl_p.arrStatusEstufas[gvl.actEst].inicioReator,'/');
gvl_p.arrStatusEstufas[gvl.actEst].inicioReator := concat(gvl_p.arrStatusEstufas[gvl.actEst].inicioReator,mes);
gvl_p.arrStatusEstufas[gvl.actEst].inicioReator := concat(gvl_p.arrStatusEstufas[gvl.actEst].inicioReator,'/');
gvl_p.arrStatusEstufas[gvl.actEst].inicioReator := concat(gvl_p.arrStatusEstufas[gvl.actEst].inicioReator,ano);

///// CALCULO DE DEFINIÇÃO SE O PROCESSO PASSA DAS 36 HORAS LIMITES ----------------------------------------
timeCalc:= (gvl_p.arrStatusEstufas[gvl.actEst].prevFimSeca - systemtime_to_dt(gvl.fbGetLocalSystemTime.systemTime));
IF timeCalc < T#24H THEN
	gvl_P.arrStatusEstufas[gvl.actEst].fimSecagem := gvl_p.arrStatusEstufas[gvl.actEst].dtInicioReator + T#24H;
END_IF

///// DECOMPOR A VARIAVEL FIM DA SECAGEM -----------------------------------------------------------------------------------------------
gvl_p.arrStatusEstufas[gvl.actEst].diaSec := MID(STR:= DT_TO_STRING(gvl_p.arrStatusEstufas[gvl.actEst].fimSecagem) , LEN:= 2, POS:=12);
gvl_p.arrStatusEstufas[gvl.actEst].mesSec := MID(STR:= DT_TO_STRING(gvl_p.arrStatusEstufas[gvl.actEst].fimSecagem), LEN:= 2, POS:=9);
gvl_p.arrStatusEstufas[gvl.actEst].anoSec := MID(STR:= DT_TO_STRING(gvl_p.arrStatusEstufas[gvl.actEst].fimSecagem), LEN:= 2, POS:=6);
gvl_p.arrStatusEstufas[gvl.actEst].horaSec := MID(STR:= DT_TO_STRING(gvl_p.arrStatusEstufas[gvl.actEst].fimSecagem), LEN:= 2, POS:=15);
gvl_p.arrStatusEstufas[gvl.actEst].minutoSec := MID(STR:= DT_TO_STRING(gvl_p.arrStatusEstufas[gvl.actEst].fimSecagem), LEN:= 2, POS:=18);

///// IMPRIMIR A HORA E A DATA DO FIM DA SECAGEM --------------------------------------------------------------------------------------------------------
gvl_p.arrStatusEstufas[gvl.actEst].statusFimSecagem := '';
gvl_p.arrStatusEstufas[gvl.actEst].statusFimSecagem := concat(gvl_p.arrStatusEstufas[gvl.actEst].statusFimSecagem,gvl_p.arrStatusEstufas[gvl.actEst].horaSec);
gvl_p.arrStatusEstufas[gvl.actEst].statusFimSecagem := concat(gvl_p.arrStatusEstufas[gvl.actEst].statusFimSecagem,':');
gvl_p.arrStatusEstufas[gvl.actEst].statusFimSecagem := concat(gvl_p.arrStatusEstufas[gvl.actEst].statusFimSecagem,gvl_p.arrStatusEstufas[gvl.actEst].minutoSec);
gvl_p.arrStatusEstufas[gvl.actEst].statusFimSecagem := concat(gvl_p.arrStatusEstufas[gvl.actEst].statusFimSecagem,' ');
gvl_p.arrStatusEstufas[gvl.actEst].statusFimSecagem := concat(gvl_p.arrStatusEstufas[gvl.actEst].statusFimSecagem,gvl_p.arrStatusEstufas[gvl.actEst].diaSec);
gvl_p.arrStatusEstufas[gvl.actEst].statusFimSecagem := concat(gvl_p.arrStatusEstufas[gvl.actEst].statusFimSecagem,'/');
gvl_p.arrStatusEstufas[gvl.actEst].statusFimSecagem := concat(gvl_p.arrStatusEstufas[gvl.actEst].statusFimSecagem,gvl_p.arrStatusEstufas[gvl.actEst].mesSec);
gvl_p.arrStatusEstufas[gvl.actEst].statusFimSecagem := concat(gvl_p.arrStatusEstufas[gvl.actEst].statusFimSecagem,'/');
gvl_p.arrStatusEstufas[gvl.actEst].statusFimSecagem := concat(gvl_p.arrStatusEstufas[gvl.actEst].statusFimSecagem,gvl_p.arrStatusEstufas[gvl.actEst].anoSec);

///// DECOMPOR A VARIAVEL FIM DA ARMAZENAGEM -------------------------------------------------------------------------------------------
gvl_p.arrStatusEstufas[gvl.actEst].diaArm := MID(STR:= DT_TO_STRING(gvl_p.arrStatusEstufas[gvl.actEst].fimArmazenagem) , LEN:= 2, POS:=12);
gvl_p.arrStatusEstufas[gvl.actEst].mesArm := MID(STR:= DT_TO_STRING(gvl_p.arrStatusEstufas[gvl.actEst].fimArmazenagem), LEN:= 2, POS:=9);
gvl_p.arrStatusEstufas[gvl.actEst].anoArm := MID(STR:= DT_TO_STRING(gvl_p.arrStatusEstufas[gvl.actEst].fimArmazenagem), LEN:= 2, POS:=6);
gvl_p.arrStatusEstufas[gvl.actEst].horaArm := MID(STR:= DT_TO_STRING(gvl_p.arrStatusEstufas[gvl.actEst].fimArmazenagem), LEN:= 2, POS:=15);
gvl_p.arrStatusEstufas[gvl.actEst].minutoArm := MID(STR:= DT_TO_STRING(gvl_p.arrStatusEstufas[gvl.actEst].fimArmazenagem), LEN:= 2, POS:=18);

///// IMPRIMIR A HORA E A DATA DO FIM DA ARMAZENAGEM -----------------------------------------------------------------------------------------------------------
gvl_p.arrStatusEstufas[gvl.actEst].statusFimArmazenagem := '';
gvl_p.arrStatusEstufas[gvl.actEst].statusFimArmazenagem := concat(gvl_p.arrStatusEstufas[gvl.actEst].statusFimArmazenagem,gvl_p.arrStatusEstufas[gvl.actEst].horaArm);
gvl_p.arrStatusEstufas[gvl.actEst].statusFimArmazenagem := concat(gvl_p.arrStatusEstufas[gvl.actEst].statusFimArmazenagem,':');
gvl_p.arrStatusEstufas[gvl.actEst].statusFimArmazenagem := concat(gvl_p.arrStatusEstufas[gvl.actEst].statusFimArmazenagem,gvl_p.arrStatusEstufas[gvl.actEst].minutoArm);
gvl_p.arrStatusEstufas[gvl.actEst].statusFimArmazenagem := concat(gvl_p.arrStatusEstufas[gvl.actEst].statusFimArmazenagem,' ');
gvl_p.arrStatusEstufas[gvl.actEst].statusFimArmazenagem := concat(gvl_p.arrStatusEstufas[gvl.actEst].statusFimArmazenagem,gvl_p.arrStatusEstufas[gvl.actEst].diaArm);
gvl_p.arrStatusEstufas[gvl.actEst].statusFimArmazenagem := concat(gvl_p.arrStatusEstufas[gvl.actEst].statusFimArmazenagem,'/');
gvl_p.arrStatusEstufas[gvl.actEst].statusFimArmazenagem := concat(gvl_p.arrStatusEstufas[gvl.actEst].statusFimArmazenagem,gvl_p.arrStatusEstufas[gvl.actEst].mesArm);
gvl_p.arrStatusEstufas[gvl.actEst].statusFimArmazenagem := concat(gvl_P.arrStatusEstufas[gvl.actEst].statusFimArmazenagem,'/');
gvl_p.arrStatusEstufas[gvl.actEst].statusFimArmazenagem := concat(gvl_P.arrStatusEstufas[gvl.actEst].statusFimArmazenagem,gvl_p.arrStatusEstufas[gvl.actEst].anoArm);

END_IF

///// GERADOR DE LOG -------------------------------------------------------------

posicaoAtual:= INT_TO_STRING(gvl.actReat);
estufaAtual:= INT_TO_STRING(gvl.actEst);
envialog:= 'Reator adicionado a posição de Nº ';
enviaLog:= concat(envialog, posicaoAtual);
enviaLog:= concat(envialog, '.');
enviaLog:= concat(envialog, ' ESTUFA ');
enviaLog:= concat(envialog, estufaAtual);
gvl.logRegister21:= envialog;

bGravarConfigPosicao_Reator:= TRUE;

END_PROGRAM

// ---- POUs/Botons/gravarConfigPosicao_Reator_2.TcPOU
PROGRAM gravarConfigPosicao_Reator_2
VAR
	bReator: BOOL;
	posicaoAtual: STRING;
	enviaLog: STRING;
	somaReator: TIME;
	timeCalc: TIME;
	
	dia: STRING;
	mes: STRING;
	ano: STRING;
	hora: STRING;
	minuto: STRING;
	
	bGravarConfigPosicao_Reator: BOOL:= FALSE;
	
	bNotificaTime: BOOL;
	estufaAtual: STRING;
END_VAR


IF gvl.actEst = 0 THEN
gvl_p.corPosReator1[gvl.actReat].cor:= 1;
ELSIF gvl.actEst = 1 THEN
	gvl_p.corPosReator2[gvl.actReat].cor:= 1;
	ELSIF gvl.actEst = 2 THEN
		gvl_p.corPosReator3[gvl.actReat].cor:= 1;
		END_IF
	

///// IMPRIMIR A HORA E A DATA DO INICIO DA SECAGEM-------------------------------

IF simIniciaProg.bSimIniciaProg THEN
gvl.progInicioReat:= DT_TO_STRING(gvl.somaTempo);
gvl_p.arrStatusEstufas[gvl.actEst].dtInicioReator:= gvl.somaTempo;
dia:= MID(STR:= gvl.progInicioReat , LEN:= 2, POS:=12);
mes:= MID(STR:= gvl.progInicioReat , LEN:= 2, POS:=9);
ano:= MID(STR:= gvl.progInicioReat , LEN:= 2, POS:=6);
hora:= MID(STR:= gvl.progInicioReat , LEN:= 2, POS:=15);
minuto:= MID(STR:= gvl.progInicioReat , LEN:= 2, POS:=18);

gvl_p.arrStatusEstufas[gvl.actEst].inicioReator := '';
gvl_p.arrStatusEstufas[gvl.actEst].inicioReator := concat(gvl_p.arrStatusEstufas[gvl.actEst].inicioReator,hora);
gvl_p.arrStatusEstufas[gvl.actEst].inicioReator := concat(gvl_p.arrStatusEstufas[gvl.actEst].inicioReator,':');
gvl_p.arrStatusEstufas[gvl.actEst].inicioReator := concat(gvl_p.arrStatusEstufas[gvl.actEst].inicioReator,minuto);
gvl_p.arrStatusEstufas[gvl.actEst].inicioReator := concat(gvl_p.arrStatusEstufas[gvl.actEst].inicioReator,' ');
gvl_p.arrStatusEstufas[gvl.actEst].inicioReator := concat(gvl_p.arrStatusEstufas[gvl.actEst].inicioReator,dia);
gvl_p.arrStatusEstufas[gvl.actEst].inicioReator := concat(gvl_p.arrStatusEstufas[gvl.actEst].inicioReator,'/');
gvl_p.arrStatusEstufas[gvl.actEst].inicioReator := concat(gvl_p.arrStatusEstufas[gvl.actEst].inicioReator,mes);
gvl_p.arrStatusEstufas[gvl.actEst].inicioReator := concat(gvl_p.arrStatusEstufas[gvl.actEst].inicioReator,'/');
gvl_p.arrStatusEstufas[gvl.actEst].inicioReator := concat(gvl_p.arrStatusEstufas[gvl.actEst].inicioReator,ano);

///// CALCULO DE DEFINIÇÃO SE O PROCESSO PASSA DAS 36 HORAS LIMITES ----------------------------------------
timeCalc:= (gvl_p.arrStatusEstufas[gvl.actEst].prevFimSeca - systemtime_to_dt(gvl.fbGetLocalSystemTime.systemTime));
IF timeCalc < T#24H THEN
	gvl_P.arrStatusEstufas[gvl.actEst].fimSecagem := gvl_p.arrStatusEstufas[gvl.actEst].dtInicioReator + T#24H;
END_IF

///// DECOMPOR A VARIAVEL FIM DA SECAGEM -----------------------------------------------------------------------------------------------
gvl_p.arrStatusEstufas[gvl.actEst].diaSec := MID(STR:= DT_TO_STRING(gvl_p.arrStatusEstufas[gvl.actEst].fimSecagem) , LEN:= 2, POS:=12);
gvl_p.arrStatusEstufas[gvl.actEst].mesSec := MID(STR:= DT_TO_STRING(gvl_p.arrStatusEstufas[gvl.actEst].fimSecagem), LEN:= 2, POS:=9);
gvl_p.arrStatusEstufas[gvl.actEst].anoSec := MID(STR:= DT_TO_STRING(gvl_p.arrStatusEstufas[gvl.actEst].fimSecagem), LEN:= 2, POS:=6);
gvl_p.arrStatusEstufas[gvl.actEst].horaSec := MID(STR:= DT_TO_STRING(gvl_p.arrStatusEstufas[gvl.actEst].fimSecagem), LEN:= 2, POS:=15);
gvl_p.arrStatusEstufas[gvl.actEst].minutoSec := MID(STR:= DT_TO_STRING(gvl_p.arrStatusEstufas[gvl.actEst].fimSecagem), LEN:= 2, POS:=18);

///// IMPRIMIR A HORA E A DATA DO FIM DA SECAGEM --------------------------------------------------------------------------------------------------------
gvl_p.arrStatusEstufas[gvl.actEst].statusFimSecagem := '';
gvl_p.arrStatusEstufas[gvl.actEst].statusFimSecagem := concat(gvl_p.arrStatusEstufas[gvl.actEst].statusFimSecagem,gvl_p.arrStatusEstufas[gvl.actEst].horaSec);
gvl_p.arrStatusEstufas[gvl.actEst].statusFimSecagem := concat(gvl_p.arrStatusEstufas[gvl.actEst].statusFimSecagem,':');
gvl_p.arrStatusEstufas[gvl.actEst].statusFimSecagem := concat(gvl_p.arrStatusEstufas[gvl.actEst].statusFimSecagem,gvl_p.arrStatusEstufas[gvl.actEst].minutoSec);
gvl_p.arrStatusEstufas[gvl.actEst].statusFimSecagem := concat(gvl_p.arrStatusEstufas[gvl.actEst].statusFimSecagem,' ');
gvl_p.arrStatusEstufas[gvl.actEst].statusFimSecagem := concat(gvl_p.arrStatusEstufas[gvl.actEst].statusFimSecagem,gvl_p.arrStatusEstufas[gvl.actEst].diaSec);
gvl_p.arrStatusEstufas[gvl.actEst].statusFimSecagem := concat(gvl_p.arrStatusEstufas[gvl.actEst].statusFimSecagem,'/');
gvl_p.arrStatusEstufas[gvl.actEst].statusFimSecagem := concat(gvl_p.arrStatusEstufas[gvl.actEst].statusFimSecagem,gvl_p.arrStatusEstufas[gvl.actEst].mesSec);
gvl_p.arrStatusEstufas[gvl.actEst].statusFimSecagem := concat(gvl_p.arrStatusEstufas[gvl.actEst].statusFimSecagem,'/');
gvl_p.arrStatusEstufas[gvl.actEst].statusFimSecagem := concat(gvl_p.arrStatusEstufas[gvl.actEst].statusFimSecagem,gvl_p.arrStatusEstufas[gvl.actEst].anoSec);

///// DECOMPOR A VARIAVEL FIM DA ARMAZENAGEM -------------------------------------------------------------------------------------------
gvl_p.arrStatusEstufas[gvl.actEst].diaArm := MID(STR:= DT_TO_STRING(gvl_p.arrStatusEstufas[gvl.actEst].fimArmazenagem) , LEN:= 2, POS:=12);
gvl_p.arrStatusEstufas[gvl.actEst].mesArm := MID(STR:= DT_TO_STRING(gvl_p.arrStatusEstufas[gvl.actEst].fimArmazenagem), LEN:= 2, POS:=9);
gvl_p.arrStatusEstufas[gvl.actEst].anoArm := MID(STR:= DT_TO_STRING(gvl_p.arrStatusEstufas[gvl.actEst].fimArmazenagem), LEN:= 2, POS:=6);
gvl_p.arrStatusEstufas[gvl.actEst].horaArm := MID(STR:= DT_TO_STRING(gvl_p.arrStatusEstufas[gvl.actEst].fimArmazenagem), LEN:= 2, POS:=15);
gvl_p.arrStatusEstufas[gvl.actEst].minutoArm := MID(STR:= DT_TO_STRING(gvl_p.arrStatusEstufas[gvl.actEst].fimArmazenagem), LEN:= 2, POS:=18);

///// IMPRIMIR A HORA E A DATA DO FIM DA ARMAZENAGEM -----------------------------------------------------------------------------------------------------------
gvl_p.arrStatusEstufas[gvl.actEst].statusFimArmazenagem := '';
gvl_p.arrStatusEstufas[gvl.actEst].statusFimArmazenagem := concat(gvl_p.arrStatusEstufas[gvl.actEst].statusFimArmazenagem,gvl_p.arrStatusEstufas[gvl.actEst].horaArm);
gvl_p.arrStatusEstufas[gvl.actEst].statusFimArmazenagem := concat(gvl_p.arrStatusEstufas[gvl.actEst].statusFimArmazenagem,':');
gvl_p.arrStatusEstufas[gvl.actEst].statusFimArmazenagem := concat(gvl_p.arrStatusEstufas[gvl.actEst].statusFimArmazenagem,gvl_p.arrStatusEstufas[gvl.actEst].minutoArm);
gvl_p.arrStatusEstufas[gvl.actEst].statusFimArmazenagem := concat(gvl_p.arrStatusEstufas[gvl.actEst].statusFimArmazenagem,' ');
gvl_p.arrStatusEstufas[gvl.actEst].statusFimArmazenagem := concat(gvl_p.arrStatusEstufas[gvl.actEst].statusFimArmazenagem,gvl_p.arrStatusEstufas[gvl.actEst].diaArm);
gvl_p.arrStatusEstufas[gvl.actEst].statusFimArmazenagem := concat(gvl_p.arrStatusEstufas[gvl.actEst].statusFimArmazenagem,'/');
gvl_p.arrStatusEstufas[gvl.actEst].statusFimArmazenagem := concat(gvl_p.arrStatusEstufas[gvl.actEst].statusFimArmazenagem,gvl_p.arrStatusEstufas[gvl.actEst].mesArm);
gvl_p.arrStatusEstufas[gvl.actEst].statusFimArmazenagem := concat(gvl_P.arrStatusEstufas[gvl.actEst].statusFimArmazenagem,'/');
gvl_p.arrStatusEstufas[gvl.actEst].statusFimArmazenagem := concat(gvl_P.arrStatusEstufas[gvl.actEst].statusFimArmazenagem,gvl_p.arrStatusEstufas[gvl.actEst].anoArm);

END_IF

///// GERADOR DE LOG -------------------------------------------------------------

posicaoAtual:= INT_TO_STRING(gvl.actReat);
estufaAtual:= INT_TO_STRING(gvl.actEst);
envialog:= 'Reator adicionado a posição de Nº ';
enviaLog:= concat(envialog, posicaoAtual);
enviaLog:= concat(envialog, '.');
enviaLog:= concat(envialog, ' ESTUFA ');
enviaLog:= concat(envialog, estufaAtual);
gvl.logRegister20:= envialog;

bGravarConfigPosicao_Reator:= TRUE;

END_PROGRAM

// ---- POUs/Botons/iniciaProgramacaoEstufa.TcPOU
PROGRAM iniciaProgramacaoEstufa
VAR
END_VAR


gvl.progInicio[gvl.actEst]:= DT_TO_STRING(gvl.somaTempo);

IF gvl.actEst = 0 THEN
	gvl.estAtiva:= '203/019';
	ELSIF gvl.actEst = 1 THEN
		gvl.estAtiva:= '203/020';
		ELSIF gvl.actEst = 2 THEN
			gvl.estAtiva:= '203/021';
END_IF

(*FOR gvl.n:=1 TO 24 BY 1 DO
	IF gvl.aPositionsE019[gvl.n].numOF <> 0 THEN
		gvl.totalPos:= gvl.totalPos + 1;
	END_IF
END_FOR*)

gvl.dia:= MID(STR:= gvl.progInicio[gvl.actEst] , LEN:= 2, POS:=12);
gvl.mes:= MID(STR:= gvl.progInicio[gvl.actEst] , LEN:= 2, POS:=9);
gvl.ano:= MID(STR:= gvl.progInicio[gvl.actEst] , LEN:= 2, POS:=6);
gvl.hora:= MID(STR:= gvl.progInicio[gvl.actEst] , LEN:= 2, POS:=15);
gvl.minuto:= MID(STR:= gvl.progInicio[gvl.actEst] , LEN:= 2, POS:=18);

END_PROGRAM

// ---- POUs/Botons/posCarrinho.TcPOU
PROGRAM posCarrinho
VAR
	timeCalc: TIME;
	bNotificaTime: BOOL:= TRUE;
END_VAR


///// CALCULO DE DEFINIÇÃO SE O PROCESSO PASSA DAS 36 HORAS LIMITES ----------------------------------------
timeCalc:= (gvl_p.arrStatusEstufas[0].prevFimSeca - systemtime_to_dt(gvl.fbGetLocalSystemTime.systemTime));
IF timeCalc < T#24H THEN
	bNotificaTime:= FALSE;
	ELSE
		bNotificaTime:= TRUE;
		
END_IF

END_PROGRAM

// ---- POUs/Botons/posCarrinho3.TcPOU
PROGRAM posCarrinho3
VAR
	timeCalc: TIME;
	bNotificaTime: BOOL:= TRUE;
END_VAR


///// CALCULO DE DEFINIÇÃO SE O PROCESSO PASSA DAS 36 HORAS LIMITES ----------------------------------------
timeCalc:= (gvl_p.arrStatusEstufas[2].prevFimSeca - systemtime_to_dt(gvl.fbGetLocalSystemTime.systemTime));
IF timeCalc < T#24H and bNotificaTime THEN
	bNotificaTime:= FALSE;
	ELSE
		bNotificaTime:= TRUE;
		
END_IF

END_PROGRAM

// ---- POUs/Botons/simIniciaProg_Manual.TcPOU
PROGRAM simIniciaProg_Manual
VAR
	bSimIniciaProg: BOOL:= FALSE;
	posicaoAtual: STRING;
	envialog: STRING;
	bGravarConfigPosicao_Reator: BOOL;
END_VAR


gvl_p.arrStatusEstufas[gvl.actEst].startManual := TRUE;

bGravarConfigPosicao_Reator:= TRUE;

END_PROGRAM

// ---- POUs/Botons/simIniciaProg_Manual_3.TcPOU
PROGRAM simIniciaProg_Manual_3
VAR
	bSimIniciaProg: BOOL:= FALSE;
	posicaoAtual: STRING;
	envialog: STRING;
	bGravarConfigPosicao_Reator: BOOL;
END_VAR


gvl_p.arrStatusEstufas[gvl.actEst].startManual := TRUE;

bGravarConfigPosicao_Reator:= TRUE;

END_PROGRAM

// ---- POUs/Botons/simIniciaProg_Manual_2.TcPOU
PROGRAM simIniciaProg_Manual_2
VAR
	bSimIniciaProg: BOOL:= FALSE;
	posicaoAtual: STRING;
	envialog: STRING;
	bGravarConfigPosicao_Reator: BOOL;
END_VAR


gvl_p.arrStatusEstufas[gvl.actEst].startManual := TRUE;

bGravarConfigPosicao_Reator:= TRUE;

END_PROGRAM

// ---- POUs/Chart_Gen.TcPOU
PROGRAM Chart_Gen
VAR
	bstart: BOOL;
	i: INT;
	temperatura1: REAL;
	temperatura2: REAL;
	j: INT;
	fbChartTime019: Ton;
	fbTimerTrigger019: R_trig;
	fbChartTime020: Ton;
	fbTimerTrigger020: R_trig;
	fbChartTime021: Ton;
	fbTimerTrigger021: R_trig;
	k: INT;
	l: INT;
	m: INT;
	n: INT;
END_VAR


fbChartTime019(in:=gvl.bstartchart019, pt:=T#10M);
fbTimerTrigger019(clk:=fbChartTime019.Q);

IF fbTimerTrigger019.Q THEN
	i:=i+1;
	IF i <= 720 THEN
	FOR j:=i TO 720 BY 1 DO
	gvl_p.arrTemp019[j]:= gvl.zona1atual_019;
	gvl_p.arrTempVisu019[j]:= gvl.zona2atual_019;
	END_FOR
	ELSE
		i:= 0;
	END_IF
	
	fbChartTime019(in:=FALSE);
END_IF

fbChartTime020(in:=gvl.bstartchart020, pt:=T#10M);
fbTimerTrigger020(clk:=fbChartTime020.Q);

IF fbTimerTrigger020.Q THEN
	k:=k+1;
	IF k <= 720 THEN
	FOR l:=k TO 720 BY 1 DO
	gvl_p.arrTemp020[l]:= gvl.zona1atual_020;
	gvl_p.arrTempVisu020[l]:= gvl.zona2atual_020;
	END_FOR
	ELSE
		k:= 0;
	END_IF
	
	fbChartTime020(in:=FALSE);
END_IF

fbChartTime021(in:=gvl.bstartchart021, pt:=T#10M);
fbTimerTrigger021(clk:=fbChartTime021.Q);

IF fbTimerTrigger021.Q THEN
	m:=m+1;
	IF m <= 720 THEN
	FOR n:=m TO 720 BY 1 DO
	gvl_p.arrTemp021[n]:= gvl.zona1atual_021;
	gvl_p.arrTempVisu021[n]:= gvl.zona2atual_021;
	END_FOR
	ELSE
		m:= 0;
	END_IF
	
	fbChartTime021(in:=FALSE);
END_IF

IF NOT gvl.bstartchart019 THEN
	i:= 0;
END_IF
IF NOT gvl.bstartchart020 THEN
	k:= 0;
END_IF
IF NOT gvl.bstartchart021 THEN
	m:= 0;
END_IF

END_PROGRAM

// ---- POUs/historical.TcPOU
PROGRAM historical
VAR
	
	state: INT;
END_VAR




CASE state OF

0:	
IF gvl.bHistory THEN
	CASE gvl.radioEstufa OF
0:
	IF gvl.radioFiltro = 0 THEN
		state:=10;
	gvl.sCmdSelect19:= 'SELECT [data],[hora],[auto],[pos],[OF],[lote],[class],[pot],[isola],[fPot],[reator],[time],[temp] FROM [dbo].[ProcessTable19] 
	WHERE data=$'';
	gvl.sCmdSelect19:= concat(gvl.sCmdSelect19,gvl.arrCVSfilter[0].ano);
	gvl.sCmdSelect19:= concat(gvl.sCmdSelect19,'-');
	gvl.sCmdSelect19:= concat(gvl.sCmdSelect19,gvl.arrCVSfilter[0].mes);
	gvl.sCmdSelect19:= concat(gvl.sCmdSelect19,'-');
	gvl.sCmdSelect19:= concat(gvl.sCmdSelect19,gvl.arrCVSfilter[0].dia);
	gvl.sCmdSelect19:= concat(gvl.sCmdSelect19,'$';');
	ELSIF gvl.radioFiltro = 1 THEN
		state:=10;
	gvl.sCmdSelect19:= 'SELECT [data],[hora],[auto],[pos],[OF],[lote],[class],[pot],[isola],[fPot],[reator],[time],[temp] FROM [dbo].[ProcessTable19] 
	WHERE OF=$'';
	gvl.sCmdSelect19:= concat(gvl.sCmdSelect19,gvl.arrCVSfilter[0].ordem);
	gvl.sCmdSelect19:= concat(gvl.sCmdSelect19,'$';');
	ELSIF gvl.radioFiltro = 2 THEN
		state:=10;
	gvl.sCmdSelect19:= 'SELECT [data],[hora],[auto],[pos],[OF],[lote],[class],[pot],[isola],[fPot],[reator],[time],[temp] FROM [dbo].[ProcessTable19] 
	WHERE lote=$'';
	gvl.sCmdSelect19:= concat(gvl.sCmdSelect19,gvl.arrCVSfilter[0].lote);
	gvl.sCmdSelect19:= concat(gvl.sCmdSelect19,'$';');
	END_IF
	
1:
	IF gvl.radioFiltro = 0 THEN
		state:=10;
	gvl.sCmdSelect19:= 'SELECT [data],[hora],[auto],[pos],[OF],[lote],[class],[pot],[isola],[fPot],[reator],[time],[temp] FROM [dbo].[ProcessTable20] 
	WHERE data=$'';
	gvl.sCmdSelect19:= concat(gvl.sCmdSelect19,gvl.arrCVSfilter[0].ano);
	gvl.sCmdSelect19:= concat(gvl.sCmdSelect19,'-');
	gvl.sCmdSelect19:= concat(gvl.sCmdSelect19,gvl.arrCVSfilter[0].mes);
	gvl.sCmdSelect19:= concat(gvl.sCmdSelect19,'-');
	gvl.sCmdSelect19:= concat(gvl.sCmdSelect19,gvl.arrCVSfilter[0].dia);
	gvl.sCmdSelect19:= concat(gvl.sCmdSelect19,'$';');
	ELSIF gvl.radioFiltro = 1 THEN
		state:=10;
	gvl.sCmdSelect19:= 'SELECT [data],[hora],[auto],[pos],[OF],[lote],[class],[pot],[isola],[fPot],[reator],[time],[temp] FROM [dbo].[ProcessTable20] 
	WHERE OF=$'';
	gvl.sCmdSelect19:= concat(gvl.sCmdSelect19,gvl.arrCVSfilter[0].ordem);
	gvl.sCmdSelect19:= concat(gvl.sCmdSelect19,'$';');
	ELSIF gvl.radioFiltro = 2 THEN
		state:=10;
	gvl.sCmdSelect19:= 'SELECT [data],[hora],[auto],[pos],[OF],[lote],[class],[pot],[isola],[fPot],[reator],[time],[temp] FROM [dbo].[ProcessTable20] 
	WHERE lote=$'';
	gvl.sCmdSelect19:= concat(gvl.sCmdSelect19,gvl.arrCVSfilter[0].lote);
	gvl.sCmdSelect19:= concat(gvl.sCmdSelect19,'$';');
	END_IF
	
2:
	IF gvl.radioFiltro = 0 THEN
		state:=10;
	gvl.sCmdSelect19:= 'SELECT [data],[hora],[auto],[pos],[OF],[lote],[class],[pot],[isola],[fPot],[reator],[time],[temp] FROM [dbo].[ProcessTable21] 
	WHERE data=$'';
	gvl.sCmdSelect19:= concat(gvl.sCmdSelect19,gvl.arrCVSfilter[0].ano);
	gvl.sCmdSelect19:= concat(gvl.sCmdSelect19,'-');
	gvl.sCmdSelect19:= concat(gvl.sCmdSelect19,gvl.arrCVSfilter[0].mes);
	gvl.sCmdSelect19:= concat(gvl.sCmdSelect19,'-');
	gvl.sCmdSelect19:= concat(gvl.sCmdSelect19,gvl.arrCVSfilter[0].dia);
	gvl.sCmdSelect19:= concat(gvl.sCmdSelect19,'$';');
	ELSIF gvl.radioFiltro = 1 THEN
		state:=10;
	gvl.sCmdSelect19:= 'SELECT [data],[hora],[auto],[pos],[OF],[lote],[class],[pot],[isola],[fPot],[reator],[time],[temp] FROM [dbo].[ProcessTable21] 
	WHERE OF=$'';
	gvl.sCmdSelect19:= concat(gvl.sCmdSelect19,gvl.arrCVSfilter[0].ordem);
	gvl.sCmdSelect19:= concat(gvl.sCmdSelect19,'$';');
	ELSIF gvl.radioFiltro = 2 THEN
		state:=10;
	gvl.sCmdSelect19:= 'SELECT [data],[hora],[auto],[pos],[OF],[lote],[class],[pot],[isola],[fPot],[reator],[time],[temp] FROM [dbo].[ProcessTable21] 
	WHERE lote=$'';
	gvl.sCmdSelect19:= concat(gvl.sCmdSelect19,gvl.arrCVSfilter[0].lote);
	gvl.sCmdSelect19:= concat(gvl.sCmdSelect19,'$';');
	END_IF
	END_CASE
ELSE
	state:=0;	
END_IF

10:
IF NOT main.bBusySelect19 THEN
	state:=20;
	gvl.bSelect19:= TRUE;
ELSE
	state:=10;
END_IF

20:
IF NOT main.bBusySelect19 THEN
	state:=30;
	gvl.bSelect19:= FALSE;
	P_TextModeWrite.bWrite:= TRUE;
ELSE
	state:=20;
END_IF

30:
IF NOT P_TextModeWrite.bBusy AND not P_TextModeWrite.bWrite THEN
	state:=0;
	gvl.bHistory:=FALSE;
ELSE
	state:=30;
END_IF

END_CASE

END_PROGRAM

// ---- POUs/MAIN.TcPOU
PROGRAM MAIN
VAR
	
	i: INT;
	temperatura: REAL;
	sDB_Operador: STRING;
	j: INT;
	login: string;
	start: BOOL;
	boot: bool;
	
	concatena: BOOL;
	barTimeSec: DWORD;
	barTimeArm: DWORD;
	bardintSec19: DINT;
	bardintArm19: DINT;
	bTravaRegressivaS19: BOOL;
	bTravaRegressivaA19: BOOL;
	l: INT;
	readAnalog: REAL;
	number: int;
	bTravaRegressivaS20: BOOL;
	bTravaRegressivaA20: bool;
	bardintSec20: UDINT;
	bardintArm20: UDINT;
	bTravaRegressivaS21: BOOL;
	bTravaRegressivaA21: BOOL;
	bardintSec21: UDINT;
	bardintArm21: UDINT;
	barTimeSec19: DWORD;
	barTimeArm19: DWORD;
	barTimeSec20: DWORD;
	barTimeArm20: DWORD;
	barTimeSec21: DWORD;
	barTimeArm21: DWORD;
	k: INT;
	nabas1: INT;
	nabas2: INT;
	nabas3: INT;
	tweet1: INT;
	tweet2: INT;
	tweet3: INT;
	manual: STRING;
	try: BOOL;
	
	CloseApp: BOOL;
    closeApplication : NT_StartProcess;
	
	fbDBRecordInsertLog : FB_DBRecordInsert_EX;
	fbDBRecordInsertProc : FB_DBRecordInsert_EX;
	fbDBRecordArraySelect19 : FB_DBRecordArraySelect;
	fbDBRecordArraySelect20 : FB_DBRecordArraySelect;
	fbDBRecordArraySelect21 : FB_DBRecordArraySelect;
	
	bBusyInsertLog: BOOL;
	bBusyInsertProc: BOOL;
	nErrIDInsertLog: UDINT;
	nErrIDInsertProc: UDINT;
	bErrorInsertLog: BOOL;
	bErrorInsertProc: BOOL;
	bSelect: BOOL;
	bBusySelect: BOOL;
	bErrorSelect: BOOL;
	nErrIDSelect: UDINT;
	nRecords: UDINT;
	
	
	envialog: STRING(INT#36);
	user: INT;
	bBusySelect19: BOOL;
	logout: DWORD;
	bBusySelect20: BOOL;
	bBusySelect21: BOOL;
	ultimoLogin: STRING;
	selo19emrg: BOOL;
	tOperador: ton;
	
	sUserLatched: STRING;
END_VAR


Chart_Gen();
registradorLog();
registradorLog20();
registradorLog21();
registerProc();
registerProc20();
registerProc21();
Rotina019();
Rotina019_Manual();
Rotina020();
Rotina020_Manual();
Rotina021();
Rotina021_Manual();
POU_Persistent();
historical();
P_TextModeWrite();(* This sample program opens and writes CSV file in text mode *)
	

gvl.somaTempo:= SYSTEMTIME_TO_DT(gvl.fbGetLocalSystemTime.systemTime);
	


// CALCULO DAS TEMPERATURAS 019 ---------------------------------------------------------------------------------------
gvl.zona1atual_019:= (INT_TO_REAL(gvl.AnalogIn_4_20[0]*200)/32767);
gvl.zona2atual_019:= (INT_TO_REAL(gvl.AnalogIn_4_20[1]*200)/32767);
gvl.zonaSegAtual_019:= (INT_TO_REAL(gvl.AnalogIn_4_20[2]*200)/32767);

gvl.AnalogOut_0_10[0]:= (gvl_p.zona1setpt_019)*164;
gvl.AnalogOut_0_10[1]:= (gvl_p.zona2setpt_019)*164;
gvl.AnalogOut_0_10[2]:= (gvl_p.zonaSegSetpt_019)*164;

// CALCULO DAS TEMPERATURAS 020 ---------------------------------------------------------------------------------------
gvl.zona1atual_020:= (INT_TO_REAL(gvl.AnalogIn_4_20[3]*200)/32767);
gvl.zona2atual_020:= (INT_TO_REAL(gvl.AnalogIn_4_20[4]*200)/32767);
gvl.zonaSegAtual_020:= (INT_TO_REAL(gvl.AnalogIn_4_20[5]*200)/32767);

gvl.AnalogOut_0_10[3]:= (gvl_p.zona1setpt_020)*164;
gvl.AnalogOut_0_10[4]:= (gvl_p.zona2setpt_020)*164;
gvl.AnalogOut_0_10[5]:= (gvl_p.zonaSegSetpt_020)*164;

// CALCULO DAS TEMPERATURAS 021 ---------------------------------------------------------------------------------------
gvl.zona1atual_021:= (INT_TO_REAL(gvl.AnalogIn_4_20[8]*200)/32767);
gvl.zona2atual_021:= (INT_TO_REAL(gvl.AnalogIn_4_20[6]*200)/32767);
gvl.zonaSegAtual_021:= (INT_TO_REAL(gvl.AnalogIn_4_20[7]*200)/32767);

gvl.AnalogOut_0_10[8]:= (gvl_p.zona1setpt_021)*164;
gvl.AnalogOut_0_10[6]:= (gvl_p.zona2setpt_021)*164;
gvl.AnalogOut_0_10[7]:= (gvl_p.zonaSegSetpt_021)*164;

// ROTINA PARA CALCULO DE QUANTIDADE DE POSIÇÕES E UTILIZADA -----------------------------------------------------------

gvl.totalPos[0]:=0;
gvl.totalPos[1]:=0;
gvl.totalPos[2]:=0;
FOR j:=1 TO 24 BY 1 DO
	IF gvl_p.aPositionsE019[j].cor = 0 THEN
		gvl.totalPos[0]:= gvl.totalPos[0];
	ELSE
		gvl.totalPos[0]:= gvl.totalPos[0]+1;
	END_IF
	
	IF gvl_p.aPositionsE020[j].cor = 0 THEN
		gvl.totalPos[1]:= gvl.totalPos[1];
	ELSE
		gvl.totalPos[1]:= gvl.totalPos[1]+1;			
	END_IF
	
	IF gvl_p.aPositionsE021[j].cor = 0 THEN
		gvl.totalPos[2]:= gvl.totalPos[2];
	ELSE
		gvl.totalPos[2]:= gvl.totalPos[2]+1;			
	END_IF
END_FOR


// VERIFICADOR DE PRESENÇA DE REATOR -----------------------------------------------------------------------------------

FOR j:=1 TO 24 BY 1 DO
	IF gvl_p.aPositionsE019[j].reator THEN
		nabas1:=nabas1;
	ELSE
		nabas1:=nabas1+1;			
	END_IF	
	
	IF nabas1 > 0 THEN
	gvl_p.bCarrinhoReator1:=FALSE;
	ELSE
		gvl_p.bCarrinhoReator1:=TRUE;
	END_IF
	
	IF gvl_p.aPositionsE020[j].reator THEN
		nabas2:=nabas2;
	ELSE
		nabas2:=nabas2+1;			
	END_IF	
	
	IF nabas2 > 0 THEN
	gvl_p.bCarrinhoReator2:=FALSE;
	ELSE
		gvl_p.bCarrinhoReator2:=TRUE;
	END_IF
	
	IF gvl_p.aPositionsE021[j].reator THEN
		nabas3:=nabas3;
	ELSE
		nabas3:=nabas3+1;			
	END_IF	
	
	IF nabas3 > 0 THEN
	gvl_p.bCarrinhoReator3:=FALSE;
	ELSE
		gvl_p.bCarrinhoReator3:=TRUE;
	END_IF
END_FOR

nabas1:=0;
nabas2:=0;
nabas3:=0;

// CALCULADOR DO TEMPO TOTAL MANUAL ----------------------------------------------------------------------------

gvl.totalManual[0]:=gvl_p.arr_CustomTime[1,1]+gvl_p.arr_CustomTime[1,2]+
					gvl_p.arr_CustomTime[1,3]+gvl_p.arr_CustomTime[1,4]+
					gvl_p.arr_CustomTime[1,5]+gvl_p.arr_CustomTime[1,6]+
					gvl_p.arr_CustomTime[1,7]+gvl_p.arr_CustomTime[1,8]+
					gvl_p.arr_CustomTime[1,9]+gvl_p.arr_CustomTime[1,10];

gvl.totalManual[1]:=gvl_p.arr_CustomTime_020[1,1]+gvl_p.arr_CustomTime_020[1,2]+
					gvl_p.arr_CustomTime_020[1,3]+gvl_p.arr_CustomTime_020[1,4]+
					gvl_p.arr_CustomTime_020[1,5]+gvl_p.arr_CustomTime_020[1,6]+
					gvl_p.arr_CustomTime_020[1,7]+gvl_p.arr_CustomTime_020[1,8]+
					gvl_p.arr_CustomTime_020[1,9]+gvl_p.arr_CustomTime_020[1,10];
					
gvl.totalManual[2]:=gvl_p.arr_CustomTime_021[1,1]+gvl_p.arr_CustomTime_021[1,2]+
					gvl_p.arr_CustomTime_021[1,3]+gvl_p.arr_CustomTime_021[1,4]+
					gvl_p.arr_CustomTime_021[1,5]+gvl_p.arr_CustomTime_021[1,6]+
					gvl_p.arr_CustomTime_021[1,7]+gvl_p.arr_CustomTime_021[1,8]+
					gvl_p.arr_CustomTime_021[1,9]+gvl_p.arr_CustomTime_021[1,10];
					
// CONTAGEM REGRESSIVA DOS TEMPOS DAS ESTUFAS --------------------------------------------------------------------------

IF gvl_p.arrStatusEstufas[0].fimSecagem <> DT#1970-1-1-0:0:0 THEN
	IF NOT bTravaRegressivaS19 THEN
		gvl.endSeca19:= gvl_p.arrStatusEstufas[0].fimSecagem - systemtime_to_dt(gvl.fbGetLocalSystemTime.systemTime);
	END_IF
	IF NOT bTravaRegressivaA19 THEN
		gvl.endArm19:= gvl_p.arrStatusEstufas[0].fimArmazenagem - systemtime_to_dt(gvl.fbGetLocalSystemTime.systemTime);
	END_IF
barTimeSec19:= TIME_TO_DWORD(gvl.endSeca19);
barTimeArm19:= TIME_TO_DWORD(gvl.endArm19);
bardintSec19:= barTimeSec19/5688;//96h limite da barra
bardintArm19:= barTimeArm19/2275;//240h limite da barra
ELSE
	main.bardintArm19:= 0;
	main.bardintSec19:= 0;
	main.barTimeArm19:= 0;
	main.barTimeSec19:= 0;
END_IF

IF gvl_p.arrStatusEstufas[1].fimSecagem <> DT#1970-1-1-0:0:0 THEN
	IF NOT bTravaRegressivaS20 THEN
		gvl.endSeca20:= gvl_p.arrStatusEstufas[1].fimSecagem - systemtime_to_dt(gvl.fbGetLocalSystemTime.systemTime);
	END_IF
	IF NOT bTravaRegressivaA20 THEN
		gvl.endArm20:= gvl_p.arrStatusEstufas[1].fimArmazenagem - systemtime_to_dt(gvl.fbGetLocalSystemTime.systemTime);
	END_IF
barTimeSec20:= TIME_TO_DWORD(gvl.endSeca20);
barTimeArm20:= TIME_TO_DWORD(gvl.endArm20);
bardintSec20:= barTimeSec20/5688;
bardintArm20:= barTimeArm20/2275;
ELSE
	main.bardintArm20:= 0;
	main.bardintSec20:= 0;
	main.barTimeArm20:= 0;
	main.barTimeSec20:= 0;
END_IF

IF gvl_p.arrStatusEstufas[2].fimSecagem <> DT#1970-1-1-0:0:0 THEN
	IF NOT bTravaRegressivaS21 THEN
		gvl.endSeca21:= gvl_p.arrStatusEstufas[2].fimSecagem - systemtime_to_dt(gvl.fbGetLocalSystemTime.systemTime);
	END_IF
	IF NOT bTravaRegressivaA21 THEN
		gvl.endArm21:= gvl_p.arrStatusEstufas[2].fimArmazenagem - systemtime_to_dt(gvl.fbGetLocalSystemTime.systemTime);
	END_IF
barTimeSec21:= TIME_TO_DWORD(gvl.endSeca21);
barTimeArm21:= TIME_TO_DWORD(gvl.endArm21);
bardintSec21:= barTimeSec21/5688;
bardintArm21:= barTimeArm21/2275;
ELSE
	main.bardintArm21:= 0;
	main.bardintSec21:= 0;
	main.barTimeArm21:= 0;
	main.barTimeSec21:= 0;
END_IF

IF gvl_p.arrStatusEstufas[0].fimSecagem = systemtime_to_dt(gvl.fbGetLocalSystemTime.systemTime) THEN
	bTravaRegressivaS19:= TRUE;
	ELSE
		bTravaRegressivaS19:= FALSE;
END_IF

IF gvl_p.arrStatusEstufas[0].fimArmazenagem = systemtime_to_dt(gvl.fbGetLocalSystemTime.systemTime) THEN
	bTravaRegressivaA19:= TRUE;
	gvl_p.arrStatusEstufas[0].fimSecagem := DT#1970-1-1-0:0:0;
	ELSE
		bTravaRegressivaA19:= FALSE;
END_IF

IF gvl_p.arrStatusEstufas[1].fimSecagem = systemtime_to_dt(gvl.fbGetLocalSystemTime.systemTime) THEN
	bTravaRegressivaS20:= TRUE;
	ELSE
		bTravaRegressivaS20:= FALSE;
END_IF

IF gvl_p.arrStatusEstufas[1].fimArmazenagem = systemtime_to_dt(gvl.fbGetLocalSystemTime.systemTime) THEN
	bTravaRegressivaA20:= TRUE;
	gvl_p.arrStatusEstufas[1].fimSecagem := DT#1970-1-1-0:0:0;
	ELSE
		bTravaRegressivaA20:= FALSE;
END_IF

IF gvl_p.arrStatusEstufas[2].fimSecagem = systemtime_to_dt(gvl.fbGetLocalSystemTime.systemTime) THEN
	bTravaRegressivaS21:= TRUE;
	ELSE
		bTravaRegressivaS21:= FALSE;
END_IF

IF gvl_p.arrStatusEstufas[2].fimArmazenagem = systemtime_to_dt(gvl.fbGetLocalSystemTime.systemTime) THEN
	bTravaRegressivaA21:= TRUE;
	gvl_p.arrStatusEstufas[2].fimSecagem := DT#1970-1-1-0:0:0;
	ELSE
		bTravaRegressivaA21:= FALSE;
END_IF

// ROTINA DE VERIFICAÇÃO DE COR --------------------------------------------------------------------------------------

FOR i:=1 TO 24 BY 1 DO
IF GVL_p.aPositionsE019[i].cor = 0 THEN
	gvl_p.aPositionsE019[i].color:= 16#FFFFFFFF;
	ELSIF gvl_p.aPositionsE019[i].cor = 1 THEN
		gvl_p.aPositionsE019[i].color:= 16#FF00C000;
		ELSIF gvl_p.aPositionsE019[i].cor = 2 THEN
		gvl_p.aPositionsE019[i].color:= 16#FFFFFF00;
END_IF

IF GVL_p.aPositionsE020[i].cor = 0 THEN
	gvl_p.aPositionsE020[i].color:= 16#FFFFFFFF;
	ELSIF gvl_p.aPositionsE020[i].cor = 1 THEN
		gvl_p.aPositionsE020[i].color:= 16#FF00C000;
		ELSIF gvl_p.aPositionsE020[i].cor = 2 THEN
		gvl_p.aPositionsE020[i].color:= 16#FFFFFF00;
END_IF

IF GVL_p.aPositionsE021[i].cor = 0 THEN
	gvl_p.aPositionsE021[i].color:= 16#FFFFFFFF;
	ELSIF gvl_p.aPositionsE021[i].cor = 1 THEN
		gvl_p.aPositionsE021[i].color:= 16#FF00C000;
		ELSIF gvl_p.aPositionsE021[i].cor = 2 THEN
		gvl_p.aPositionsE021[i].color:= 16#FFFFFF00;
END_IF
END_FOR

FOR l:=1 TO 6 BY 1 DO
	IF GVL_p.corPosReator1[l].cor = 0 THEN
	GVL_p.corPosReator1[l].color:= 16#FFFFFFFF;
	ELSIF GVL_p.corPosReator1[l].cor = 1 THEN
		GVL_p.corPosReator1[l].color:= 16#FF00C000;
	END_IF
		
	IF GVL_p.corPosReator2[l].cor = 0 THEN
	GVL_p.corPosReator2[l].color:= 16#FFFFFFFF;
	ELSIF GVL_p.corPosReator2[l].cor = 1 THEN
		GVL_p.corPosReator2[l].color:= 16#FF00C000;
	END_IF
	
	IF GVL_p.corPosReator3[l].cor = 0 THEN
	GVL_p.corPosReator3[l].color:= 16#FFFFFFFF;
	ELSIF GVL_p.corPosReator3[l].cor = 1 THEN
		GVL_p.corPosReator3[l].color:= 16#FF00C000;
	END_IF
END_FOR

// ROTINA SYSTEM DATE TIME ---------------------------------------------------------------------------------------------

gvl.fbGetLocalSystemTime(
sNetID:= ,
bEnable:= TRUE,
dwCycle:= 1,
dwOpt:= ,
tTimeout:= ,
bValid=> ,
systemTime=> ,
tzID=> );

gvl.sSystemDateTime := systemtime_to_string(gvl.fbGetLocalSystemTime.systemTime);
gvl.sSystemDate:= MID(STR:= gvl.sSystemDateTime , LEN:= 10, POS:=1 );
gvl.sSystemTime:= MID(STR:= gvl.sSystemDateTime , LEN:= 8, POS:=12 );

// ROTINA DE SEGURANÇA -----------------------------------------------------------------------------------------------------
IF gvl.zona1atual_019 > gvl_p.zonaSegSetpt_019 OR gvl.zona2atual_019 > gvl_p.zonaSegSetpt_019 OR NOT gvl.inEmergencia019 OR NOT boot THEN
	gvl.emergencia019:= TRUE;
	gvl.pwEmerg_019:= TRUE;
	gvl.emergency:= TRUE;
	selo19emrg:= FALSE;
	boot:= TRUE;
	envialog:= 'Emergência Ativada - Estufa 019';
	gvl.logRegister19:= envialog;
END_IF

IF gvl.zona1atual_020 > gvl_p.zonaSegSetpt_020 OR gvl.zona2atual_020 > gvl_p.zonaSegSetpt_020 OR NOT gvl.inEmergencia020 OR NOT boot THEN
	gvl.emergencia020:= TRUE;
	gvl.pwEmerg_020:= TRUE;
	gvl.emergency:= TRUE;
	boot:= TRUE;
	envialog:= 'Emergência Ativada - Estufa 020';
	gvl.logRegister20:= envialog;
END_IF

IF gvl.zona1atual_021 > gvl_p.zonaSegSetpt_021 OR gvl.zona2atual_021 > gvl_p.zonaSegSetpt_021 OR NOT gvl.inEmergencia021 or not boot THEN
	gvl.emergencia021:= TRUE;
	gvl.pwEmerg_021:= TRUE;
	gvl.emergency:= TRUE;
	boot:= TRUE;
	envialog:= 'Emergência Ativada - Estufa 021';
	gvl.logRegister21:= envialog;
END_IF

//Rotina envio sinal de produção ProdWin -------------------------------------------------------------------------
IF gvl_p.etapa_process[0] = 'Secagem' THEN
	gvl.pwProd_019:= TRUE;
	ELSE
		gvl.pwProd_019:= FALSE;
END_IF

IF gvl_p.etapa_process[1] = 'Secagem' THEN
	gvl.pwProd_020:= TRUE;
	ELSE
		gvl.pwProd_020:= FALSE;
END_IF

IF gvl_p.etapa_process[2] = 'Secagem' THEN
	gvl.pwProd_021:= TRUE;
	ELSE
		gvl.pwProd_021:= FALSE;
END_IF

// SQL communication ---------------------------------------------------------------------------------------------


IF bBusyInsertLog THEN
gvl.bInsertLog:= FALSE;
END_IF
	
fbDBRecordInsertLog(
	sNetID 		:= '',
	hDBID 		:= 1,
	pCmdAddr 	:= ADR(gvl.sCmdInsertLog),
	cbCmdSize 	:= SIZEOF(gvl.sCmdInsertLog),
	bExecute 	:= gvl.bInsertLog,
	tTimeout 	:= T#3S,
	bBusy 		=> bBusyInsertLog,
	bError 		=> bErrorInsertLog,
	nErrID 		=> nErrIDInsertLog);
	
IF bBusyInsertProc THEN
gvl.bInsertProc:= FALSE;
END_IF
	
fbDBRecordInsertProc(
	sNetID 		:= '',
	hDBID 		:= 1,
	pCmdAddr 	:= ADR(gvl.sCmdInsertProc),
	cbCmdSize 	:= SIZEOF(gvl.sCmdInsertProc),
	bExecute 	:= gvl.bInsertProc,
	tTimeout 	:= T#3S,
	bBusy 		=> bBusyInsertProc,
	bError 		=> bErrorInsertProc,
	nErrID 		=> nErrIDInsertProc);
	

IF bBusySelect19 THEN
gvl.bSelect19:= FALSE;
END_IF

fbDBRecordArraySelect19(
	sNetID 				:= '',
	hDBID 				:= 1,
	pCmdAddr 			:= ADR(gvl.sCmdSelect19),
	cbCmdSize 			:= SIZEOF(gvl.sCmdSelect19),
	nStartIndex 		:= 0,
	nRecordCount 		:= MAX_CSV_ROWS,
	pDestAddr 			:= ADR(gvl.aSelect19),
	cbRecordArraySize 	:= SIZEOF(gvl.aSelect19),
	bExecute 			:= gvl.bSelect19,
	tTimeout 			:= T#30S,
	bBusy 				=> bBusySelect19,
	bError 				=> bErrorSelect,
	nErrID 				=> nErrIDSelect,
	nRecords 			=> nRecords,);
	
// VERIFICADOR DE LOGIN DE USUÁRIO ------------------------------------------------------------------------------------------

sDB_Operador:= WSTRING_TO_STRING(VisuElems.CurrentFullUserName);

IF sDB_Operador <> '' THEN
    sUserLatched := sDB_Operador;
END_IF

IF sUserLatched <> '' AND sUserLatched <> ultimoLogin THEN
	user:=10;
	ultimoLogin:='';
	ultimoLogin:= sUserLatched;
	tOperador(in:= TRUE, pt:=T#1S);
	envialog:= 'Usuário ';
	envialog:= concat(envialog, sUserLatched);
	envialog:= concat(envialog, ' Logado.');
	gvl.logRegister19:= envialog;
	gvl.logRegister20:= envialog;
	gvl.logRegister21:= envialog;

END_IF


// LOGICA HISTORICO ------------------------------------------------------------------------------------------------
IF gvl.radioFiltro = 0 THEN
	gvl.radioData:= FALSE;
	ELSE
		gvl.radioData:= TRUE;
END_IF

IF gvl.radioFiltro = 1 THEN
	gvl.radioOF:= FALSE;
	ELSE
		gvl.radioOF:= TRUE;
END_IF

IF gvl.radioFiltro = 2 THEN
	gvl.radioLote:= FALSE;
	ELSE
		gvl.radioLote:= TRUE;
END_IF

// LINK DE VARIAVEIS COM IOs ESTUFA 019 ------------------------------------------------------------------------------------

	gvl.sobrecarga_M1_vent_019:= gvl.DigitalIn1[1];
	gvl.sobrecarga_M2_vent_019:= gvl.DigitalIn1[2];
	gvl.sobrecarga_Purga_019:= gvl.DigitalIn1[4];
	gvl.falhaTempHigh_019:= gvl.DigitalIn1[6];
	gvl.queimador1_block_019:= gvl.DigitalIn1[8];
	gvl.queimador2_block_019:= gvl.DigitalIn1[10];
	gvl.ventilacao_Ligada_019:= gvl.DigitalIn1[12];
	gvl.aquecimento_Desligado_019:= gvl.DigitalIn1[3];
	gvl.aquecimento_Ligado_019:= gvl.DigitalIn1[5];
	gvl.fimCicloAquecimento_019:= gvl.DigitalIn1[7];
	gvl.purgandoCamara_019:= gvl.DigitalIn1[9];
	gvl.inEmergencia019:= gvl.DigitalIn3[14];
	gvl.DigitalOut1[7]:= gvl.liga_ventilacao_019;
	gvl.DigitalOut1[8]:= gvl.liga_aquecimento_019;
	gvl.DigitalOut1[9]:= gvl.desl_aquecimento_019;
	gvl.DigitalOut2[9]:= gvl.emergencia019;
	

// LINK DE VARIAVEIS COM IOs ESTUFA 020 ------------------------------------------------------------------------------------

	gvl.sobrecarga_M1_vent_020:= gvl.DigitalIn1[13];
	gvl.sobrecarga_M2_vent_020:= gvl.DigitalIn1[14];
	gvl.sobrecarga_Purga_020:= gvl.DigitalIn1[15];
	gvl.falhaTempHigh_020:= gvl.DigitalIn2[2];
	gvl.queimador1_block_020:= gvl.DigitalIn2[4];
	gvl.queimador2_block_020:= gvl.DigitalIn2[6];
	gvl.ventilacao_Ligada_020:= gvl.DigitalIn2[8];
	gvl.aquecimento_Desligado_020:= gvl.DigitalIn1[15];
	gvl.aquecimento_Ligado_020:= gvl.DigitalIn2[1];
	gvl.fimCicloAquecimento_020:= gvl.DigitalIn2[3];
	gvl.purgandoCamara_020:= gvl.DigitalIn2[5];
	gvl.inEmergencia020:= gvl.DigitalIn3[15];
	gvl.DigitalOut1[12]:= gvl.liga_ventilacao_020;
	gvl.DigitalOut1[11]:= gvl.liga_aquecimento_020;
	gvl.DigitalOut1[10]:= gvl.desl_aquecimento_020;
	gvl.DigitalOut2[10]:= gvl.emergencia020;
	

// LINK DE VARIAVEIS COM IOs ESTUFA 021 ------------------------------------------------------------------------------------

	gvl.sobrecarga_M1_vent_021:= gvl.DigitalIn2[9];
	gvl.sobrecarga_M2_vent_021:= gvl.DigitalIn2[10];
	gvl.sobrecarga_Purga_021:= gvl.DigitalIn2[12];
	gvl.falhaTempHigh_021:= gvl.DigitalIn2[14];
	gvl.queimador1_block_021:= gvl.DigitalIn2[16];
	gvl.queimador2_block_021:= gvl.DigitalIn3[2];
	gvl.ventilacao_Ligada_021:= gvl.DigitalIn3[4];
	gvl.aquecimento_Desligado_021:= gvl.DigitalIn2[11];
	gvl.aquecimento_Ligado_021:= gvl.DigitalIn2[13];
	gvl.fimCicloAquecimento_021:= gvl.DigitalIn2[15];
	gvl.purgandoCamara_021:= gvl.DigitalIn3[1];
	gvl.inEmergencia021:= gvl.DigitalIn3[16];
	gvl.DigitalOut1[13]:= gvl.liga_ventilacao_021;
	gvl.DigitalOut1[14]:= gvl.liga_aquecimento_021;
	gvl.DigitalOut1[15]:= gvl.desl_aquecimento_021;
	gvl.DigitalOut2[11]:= gvl.emergencia021;
	

// LINK DE VARIAVEIS OI PRODWIN --------------------------------------------------------------------------

	gvl.DigitalOut1[1]:= gvl.pwProd_019;
	gvl.DigitalOut1[2]:= gvl.pwEmerg_019;
	gvl.DigitalOut1[3]:= gvl.pwProd_020;
	gvl.DigitalOut1[4]:= gvl.pwEmerg_020;
	gvl.DigitalOut1[5]:= gvl.pwProd_021;
	gvl.DigitalOut1[6]:= gvl.pwEmerg_021;

END_PROGRAM

// ---- POUs/registradorLog.TcPOU
PROGRAM registradorLog
VAR
	i: INT;
	j: INT;
	k: INT;
END_VAR


IF gvl.logRegister19 <> '' THEN
	FOR i:=100 TO 1 BY -1 DO
		IF gvl_p.arrLogEstufa19[i] <> '' THEN
			gvl_p.arrLogEstufa19[i+1]:= gvl_p.arrLogEstufa19[i];
			gvl_p.arrLogEstufa19[i]:= '';
		END_IF
	END_FOR
	gvl_p.arrLogEstufa19[1]:= concat(gvl_p.arrLogEstufa19[1],gvl.sSystemDateTime);
	gvl_p.arrLogEstufa19[1]:= concat(gvl_p.arrLogEstufa19[1],'    ');
	gvl_p.arrLogEstufa19[1]:= concat(gvl_p.arrLogEstufa19[1],gvl.logRegister19);
	gvl.sCmdInsertLog:= 'INSERT INTO [dbo].[LogGeneral] ([HistoricalTime],[Description])VALUES($'$',$'$')';
	gvl.sCmdInsertLog:= insert(gvl.sCmdInsertLog,gvl.logRegister19,74);	
	gvl.sCmdInsertLog:= insert(gvl.sCmdInsertLog,gvl.sSystemDateTime,71);
	gvl.bInsertLog:=true;
	gvl.logRegister19:= '';
	
	
END_IF

END_PROGRAM

// ---- POUs/registradorLog20.TcPOU
PROGRAM registradorLog20
VAR
	i: INT;
	j: INT;
	k: INT;
END_VAR


IF gvl.logRegister20 <> '' THEN
	FOR i:=100 TO 1 BY -1 DO
		IF gvl_p.arrLogEstufa20[i] <> '' THEN
			gvl_p.arrLogEstufa20[i+1]:= gvl_p.arrLogEstufa20[i];
			gvl_p.arrLogEstufa20[i]:= '';
		END_IF
	END_FOR
	gvl_p.arrLogEstufa20[1]:= concat(gvl_p.arrLogEstufa20[1],gvl.sSystemDateTime);
	gvl_p.arrLogEstufa20[1]:= concat(gvl_p.arrLogEstufa20[1],'    ');
	gvl_p.arrLogEstufa20[1]:= concat(gvl_p.arrLogEstufa20[1],gvl.logRegister20);
	gvl.sCmdInsertLog:= 'INSERT INTO [dbo].[LogGeneral] ([HistoricalTime],[Description])VALUES($'$',$'$')';
	gvl.sCmdInsertLog:= insert(gvl.sCmdInsertLog,gvl.logRegister20,74);	
	gvl.sCmdInsertLog:= insert(gvl.sCmdInsertLog,gvl.sSystemDateTime,71);
	gvl.bInsertLog:=true;
	gvl.logRegister20:= '';
	
	
END_IF

END_PROGRAM

// ---- POUs/registradorLog21.TcPOU
PROGRAM registradorLog21
VAR
	i: INT;
	j: INT;
	k: INT;
END_VAR


IF gvl.logRegister21 <> '' THEN
	FOR i:=100 TO 1 BY -1 DO
		IF gvl_p.arrLogEstufa21[i] <> '' THEN
			gvl_p.arrLogEstufa21[i+1]:= gvl_p.arrLogEstufa21[i];
			gvl_p.arrLogEstufa21[i]:= '';
		END_IF
	END_FOR
	gvl_p.arrLogEstufa21[1]:= concat(gvl_p.arrLogEstufa21[1],gvl.sSystemDateTime);
	gvl_p.arrLogEstufa21[1]:= concat(gvl_p.arrLogEstufa21[1],'    ');
	gvl_p.arrLogEstufa21[1]:= concat(gvl_p.arrLogEstufa21[1],gvl.logRegister21);
	gvl.sCmdInsertLog:= 'INSERT INTO [dbo].[LogGeneral] ([HistoricalTime],[Description])VALUES($'$',$'$')';
	gvl.sCmdInsertLog:= insert(gvl.sCmdInsertLog,gvl.logRegister21,74);	
	gvl.sCmdInsertLog:= insert(gvl.sCmdInsertLog,gvl.sSystemDateTime,71);
	gvl.bInsertLog:=true;
	gvl.logRegister21:= '';
	
	
END_IF

END_PROGRAM

// ---- POUs/registerProc.TcPOU
PROGRAM registerProc
VAR
	i: INT;
	tempo: ton;
	state: INT;
	user: string;
END_VAR

tempo();

CASE state OF
	
0:
IF gvl_p.etapa_process[0] = 'Secagem' OR gvl_p.etapa_process[0] = 'T1' THEN
	state:=10;
	tempo(in:=TRUE, pt:=T#30M);
ELSE
	state:=0;
END_IF

10:
IF tempo.Q THEN
	state:= 20;
IF i=1 THEN
gvl.permanencia[1]:= gvl.permanencia[1]+tempo.PT;
user:= main.sDB_Operador;
END_IF
IF gvl_p.aPositionsE019[i].reator THEN
	gvl.sReator:= 'SIM';
	else
		gvl.sReator:= 'NÃO';
END_IF
if gvl_p.aPositionsE019[i].FP = 1 then
	gvl.sFp:= 'NORMAL';
	ELSIF gvl_p.aPositionsE019[i].FP = 2 THEN
		gvl.sFp:= 'REDUZIDO';
END_IF
IF gvl_p.aPositionsE019[i].isolamento = 1 THEN
	gvl.sIso:= '15';
	ELSIF gvl_p.aPositionsE019[i].isolamento = 2 THEN
		gvl.sIso:= '24';
		ELSIF gvl_p.aPositionsE019[i].isolamento = 3 THEN
			gvl.sIso:= '36';
END_IF
IF gvl_p.arrStatusEstufas[0].start THEN
	gvl.sAuto:= 'Auto';
	ELSIF gvl_p.arrStatusEstufas[0].startManual THEN
		gvl.sAuto:= 'Manu';
END_IF

gvl.sCmdInsertProc:= 'INSERT INTO [dbo].[ProcessTable19] ([data],[hora],[auto],[user],[pos],[OF],[lote],[class],[pot],[isola],[fPot],[reator],[TIME],[temp])
	VALUES ($'$',$'$',$'$',$'$',$'$',$'$',$'$',,,$'$',$'$',$'$',$'$',)';
gvl.sCmdInsertProc:= insert(gvl.sCmdInsertProc,REAL_TO_STRING(gvl.zona1atual_019),180);
gvl.sCmdInsertProc:= insert(gvl.sCmdInsertProc,TIME_TO_STRING(gvl.permanencia[1]),178);
gvl.sCmdInsertProc:= insert(gvl.sCmdInsertProc,gvl.sReator,175);
gvl.sCmdInsertProc:= insert(gvl.sCmdInsertProc,gvl.sFp,172);
gvl.sCmdInsertProc:= insert(gvl.sCmdInsertProc,gvl.sIso,169);
gvl.sCmdInsertProc:= insert(gvl.sCmdInsertProc,REAL_TO_STRING(gvl_p.aPositionsE019[i].pot),167);
gvl.sCmdInsertProc:= insert(gvl.sCmdInsertProc,REAL_TO_STRING(gvl_p.aPositionsE019[i].class),166);
gvl.sCmdInsertProc:= insert(gvl.sCmdInsertProc,gvl_p.aPositionsE019[i].lote,164);
gvl.sCmdInsertProc:= insert(gvl.sCmdInsertProc,gvl_p.aPositionsE019[i].numOF,161);
gvl.sCmdInsertProc:= insert(gvl.sCmdInsertProc,INT_TO_STRING(i),158);
gvl.sCmdInsertProc:= insert(gvl.sCmdInsertProc,user,155);
gvl.sCmdInsertProc:= insert(gvl.sCmdInsertProc,gvl.sAuto,152);
gvl.sCmdInsertProc:= insert(gvl.sCmdInsertProc,gvl.sSystemTime,149);
gvl.sCmdInsertProc:= insert(gvl.sCmdInsertProc,gvl.sSystemDate,146);

gvl.bInsertProc:= TRUE;
ELSE
	state:=10;
END_IF

20:
IF i<=24 AND NOT main.bBusyInsertProc THEN
	state:=10;
	i:=i+1;
ELSIF i=24 THEN
	state:=0;
	i:=1;
	tempo(in:=FALSE);
ELSE
	state:=20;
END_IF

END_CASE

END_PROGRAM

// ---- POUs/registerProc20.TcPOU
PROGRAM registerProc20
VAR
	i: INT;
	tempo: ton;
	state: INT;
	user: string;
END_VAR

tempo();

CASE state OF
	
0:
IF gvl_p.etapa_process[1] = 'Secagem' or gvl_p.etapa_process[1] = 'T1' THEN
	state:=10;
	tempo(in:=TRUE, pt:=T#30M);
ELSE
	state:=0;
END_IF

10:
IF tempo.Q THEN
	state:= 20;
IF i=1 THEN
gvl.permanencia[2]:= gvl.permanencia[2]+tempo.PT;
user:= main.sDB_Operador;
END_IF
IF gvl_p.aPositionsE020[i].reator THEN
	gvl.sReator:= 'SIM';
	else
		gvl.sReator:= 'NÃO';
END_IF
IF gvl_p.aPositionsE020[i].FP = 1 THEN
	gvl.sFp:= 'NORMAL';
	ELSIF gvl_p.aPositionsE020[i].FP = 2 THEN
		gvl.sFp:= 'REDUZIDO';
END_IF
IF gvl_p.aPositionsE020[i].isolamento = 1 THEN
	gvl.sIso:= '15';
	ELSIF gvl_p.aPositionsE020[i].isolamento = 2 THEN
		gvl.sIso:= '24';
		ELSIF gvl_p.aPositionsE020[i].isolamento = 3 THEN
			gvl.sIso:= '36';
END_IF
IF gvl_p.arrStatusEstufas[1].start THEN
	gvl.sAuto:= 'Auto';
	ELSIF gvl_p.arrStatusEstufas[1].startManual THEN
		gvl.sAuto:= 'Manu';
END_IF

gvl.sCmdInsertProc:= 'INSERT INTO [dbo].[ProcessTable20] ([data],[hora],[auto],[user],[pos],[OF],[lote],[class],[pot],[isola],[fPot],[reator],[TIME],[temp])
	VALUES ($'$',$'$',$'$',$'$',$'$',$'$',$'$',,,$'$',$'$',$'$',$'$',)';
gvl.sCmdInsertProc:= insert(gvl.sCmdInsertProc,REAL_TO_STRING(gvl.zona1atual_020),180);
gvl.sCmdInsertProc:= insert(gvl.sCmdInsertProc,TIME_TO_STRING(gvl.permanencia[2]),178);
gvl.sCmdInsertProc:= insert(gvl.sCmdInsertProc,gvl.sReator,175);
gvl.sCmdInsertProc:= insert(gvl.sCmdInsertProc,gvl.sFp,172);
gvl.sCmdInsertProc:= insert(gvl.sCmdInsertProc,gvl.sIso,169);
gvl.sCmdInsertProc:= insert(gvl.sCmdInsertProc,REAL_TO_STRING(gvl_p.aPositionsE020[i].pot),167);
gvl.sCmdInsertProc:= insert(gvl.sCmdInsertProc,REAL_TO_STRING(gvl_p.aPositionsE020[i].class),166);
gvl.sCmdInsertProc:= insert(gvl.sCmdInsertProc,gvl_p.aPositionsE020[i].lote,164);
gvl.sCmdInsertProc:= insert(gvl.sCmdInsertProc,gvl_p.aPositionsE020[i].numOF,161);
gvl.sCmdInsertProc:= insert(gvl.sCmdInsertProc,INT_TO_STRING(i),158);
gvl.sCmdInsertProc:= insert(gvl.sCmdInsertProc,user,155);
gvl.sCmdInsertProc:= insert(gvl.sCmdInsertProc,gvl.sAuto,152);
gvl.sCmdInsertProc:= insert(gvl.sCmdInsertProc,gvl.sSystemTime,149);
gvl.sCmdInsertProc:= insert(gvl.sCmdInsertProc,gvl.sSystemDate,146);

gvl.bInsertProc:= TRUE;
ELSE
	state:=10;
END_IF

20:
IF i<=24 AND NOT main.bBusyInsertProc THEN
	state:=10;
	i:=i+1;
ELSIF i=24 THEN
	state:=0;
	i:=1;
	tempo(in:=FALSE);
ELSE
	state:=20;
END_IF

END_CASE

END_PROGRAM

// ---- POUs/registerProc21.TcPOU
PROGRAM registerProc21
VAR
	i: INT;
	tempo: ton;
	state: INT;
	user: string;
END_VAR

tempo();

CASE state OF
	
0:
IF gvl_p.etapa_process[2] = 'Secagem' or gvl_p.etapa_process[2] = 'T1' THEN
	state:=10;
	tempo(in:=TRUE, pt:=T#30M);
ELSE
	state:=0;
END_IF

10:
IF tempo.Q THEN
	state:= 20;
IF i=1 THEN
gvl.permanencia[3]:= gvl.permanencia[3]+tempo.PT;
user:= main.sDB_Operador;
END_IF
IF gvl_p.aPositionsE021[i].reator THEN
	gvl.sReator:= 'SIM';
	else
		gvl.sReator:= 'NÃO';
END_IF
IF gvl_p.aPositionsE021[i].FP = 1 THEN
	gvl.sFp:= 'NORMAL';
	ELSIF gvl_p.aPositionsE021[i].FP = 2 THEN
		gvl.sFp:= 'REDUZIDO';
END_IF
IF gvl_p.aPositionsE021[i].isolamento = 1 THEN
	gvl.sIso:= '15';
	ELSIF gvl_p.aPositionsE021[i].isolamento = 2 THEN
		gvl.sIso:= '24';
		ELSIF gvl_p.aPositionsE021[i].isolamento = 3 THEN
			gvl.sIso:= '36';
END_IF
IF gvl_p.arrStatusEstufas[2].start THEN
	gvl.sAuto:= 'Auto';
	ELSIF gvl_p.arrStatusEstufas[2].startManual THEN
		gvl.sAuto:= 'Manu';
END_IF

gvl.sCmdInsertProc:= 'INSERT INTO [dbo].[ProcessTable21] ([data],[hora],[auto],[user],[pos],[OF],[lote],[class],[pot],[isola],[fPot],[reator],[TIME],[temp])
	VALUES ($'$',$'$',$'$',$'$',$'$',$'$',$'$',,,$'$',$'$',$'$',$'$',)';
gvl.sCmdInsertProc:= insert(gvl.sCmdInsertProc,REAL_TO_STRING(gvl.zona1atual_021),180);
gvl.sCmdInsertProc:= insert(gvl.sCmdInsertProc,TIME_TO_STRING(gvl.permanencia[3]),178);
gvl.sCmdInsertProc:= insert(gvl.sCmdInsertProc,gvl.sReator,175);
gvl.sCmdInsertProc:= insert(gvl.sCmdInsertProc,gvl.sFp,172);
gvl.sCmdInsertProc:= insert(gvl.sCmdInsertProc,gvl.sIso,169);
gvl.sCmdInsertProc:= insert(gvl.sCmdInsertProc,REAL_TO_STRING(gvl_p.aPositionsE021[i].pot),167);
gvl.sCmdInsertProc:= insert(gvl.sCmdInsertProc,REAL_TO_STRING(gvl_p.aPositionsE021[i].class),166);
gvl.sCmdInsertProc:= insert(gvl.sCmdInsertProc,gvl_p.aPositionsE021[i].lote,164);
gvl.sCmdInsertProc:= insert(gvl.sCmdInsertProc,gvl_p.aPositionsE021[i].numOF,161);
gvl.sCmdInsertProc:= insert(gvl.sCmdInsertProc,INT_TO_STRING(i),158);
gvl.sCmdInsertProc:= insert(gvl.sCmdInsertProc,user,155);
gvl.sCmdInsertProc:= insert(gvl.sCmdInsertProc,gvl.sAuto,152);
gvl.sCmdInsertProc:= insert(gvl.sCmdInsertProc,gvl.sSystemTime,149);
gvl.sCmdInsertProc:= insert(gvl.sCmdInsertProc,gvl.sSystemDate,146);

gvl.bInsertProc:= TRUE;
ELSE
	state:=10;
END_IF

20:
IF i<=24 AND NOT main.bBusyInsertProc THEN
	state:=10;
	i:=i+1;
ELSIF i=24 THEN
	state:=0;
	i:=1;
	tempo(in:=FALSE);
ELSE
	state:=20;
END_IF

END_CASE

END_PROGRAM

// ---- POUs/Rotina019.TcPOU
PROGRAM Rotina019
VAR
	status: INT;
	
	posicaoAtual: STRING;
	envialog: STRING;
	
	fbTimeVentila: ton;
	fbTimeAqueci: ton;
	
END_VAR

fbTimeVentila();
fbTimeAqueci();

CASE status OF

0:
IF gvl_p.arrStatusEstufas[0].start AND STRING_TO_DT(gvl.progInicio[0]) <= systemtime_to_dt(gvl.fbGetLocalSystemTime.systemTime)  THEN
	status:= 5;
	
	gvl.bstartchart019:= TRUE;
	gvl_p.zona1setpt_019:= gvl_p.arrStatusEstufas[0].tempSeca;
	gvl_p.zona2setpt_019:= gvl_p.arrStatusEstufas[0].tempSeca;
	gvl.liga_ventilacao_019:= TRUE;
	fbTimeVentila(in:= TRUE, pt:=T#1S);

///// GERADOR DE LOG -------------------------------------------------------------

envialog:= 'Inicializando Programação ESTUFA 019';
gvl.logRegister19:= envialog;

	gvl_p.etapa_process[0] := 'Inicializando';
	
ELSE
	status:= 0;
	IF gvl_p.arrStatusEstufas[0].start THEN
		gvl_p.etapa_process[0] := gvl.progInicio[0];
	END_IF
END_IF

5:
IF fbTimeVentila.Q THEN
	status:= 10;
	gvl.liga_ventilacao_019:=FALSE;
	fbTimeVentila(in:= FALSE);
ELSE
	status:= 5;
END_IF

10:
IF gvl.ventilacao_Ligada_019 THEN
	status:= 15;
	
	gvl.liga_aquecimento_019:= TRUE;
	fbTimeAqueci(in:= TRUE, pt:= T#1S);
	
///// GERADOR DE LOG -------------------------------------------------------------

envialog:= 'Aquecendo ESTUFA 019';
gvl.logRegister19:= envialog;
	
	gvl_p.etapa_process[0] := 'Aquecendo';
	
ELSE
	status:= 10;
END_IF

15:
IF fbTimeAqueci.Q THEN
	status:= 20;
	
	gvl.liga_aquecimento_019:= FALSE;
	fbTimeAqueci(in:=false);
ELSE
	status:= 15;
END_IF

20:
IF gvl.zona1atual_019 >= gvl_p.zona1setpt_019 THEN
	status:= 30;
	
gvl.progInicio[0]:= DT_TO_STRING(gvl.somaTempo);
	
///// CALCULAR FIM DA SECAGEM E DA ARMAZENAGEM --------------------------------------------------------------------------------
gvl_p.arrStatusEstufas[0].inicioSecagem := STRING_TO_DT(gvl.progInicio[0]);
gvl_p.arrStatusEstufas[0].fimSecagem := STRING_TO_DT(gvl.progInicio[0]) + gvl_p.arrStatusEstufas[0].tempoSecagem;
gvl_P.arrStatusEstufas[0].prevFimSeca := gvl_p.arrStatusEstufas[0].fimSecagem;
gvl_p.arrStatusEstufas[0].fimArmazenagem := gvl_p.arrStatusEstufas[0].fimSecagem + gvl_p.arrStatusEstufas[0].tempoArmazenagem ;

///// IMPRIMIR A HORA E A DATA DO INICIO DA SECAGEM ---------------------------------------------------------------------------
gvl_p.arrStatusEstufas[0].statusInicioSecagem := '';
gvl_p.arrStatusEstufas[0].statusInicioSecagem := concat(gvl_p.arrStatusEstufas[0].statusInicioSecagem,gvl.hora);
gvl_p.arrStatusEstufas[0].statusInicioSecagem := concat(gvl_p.arrStatusEstufas[0].statusInicioSecagem,':');
gvl_p.arrStatusEstufas[0].statusInicioSecagem := concat(gvl_p.arrStatusEstufas[0].statusInicioSecagem,gvl.minuto);
gvl_p.arrStatusEstufas[0].statusInicioSecagem := concat(gvl_p.arrStatusEstufas[0].statusInicioSecagem,' ');
gvl_p.arrStatusEstufas[0].statusInicioSecagem := concat(gvl_p.arrStatusEstufas[0].statusInicioSecagem,gvl.dia);
gvl_p.arrStatusEstufas[0].statusInicioSecagem := concat(gvl_p.arrStatusEstufas[0].statusInicioSecagem,'/');
gvl_p.arrStatusEstufas[0].statusInicioSecagem := concat(gvl_p.arrStatusEstufas[0].statusInicioSecagem,gvl.mes);
gvl_p.arrStatusEstufas[0].statusInicioSecagem := concat(gvl_p.arrStatusEstufas[0].statusInicioSecagem,'/');
gvl_p.arrStatusEstufas[0].statusInicioSecagem := concat(gvl_p.arrStatusEstufas[0].statusInicioSecagem,gvl.ano);

//--------------------REATOR------------------------------------

IF gravarConfigPosicao_Reator.bGravarConfigPosicao_Reator THEN
	gvl_p.arrStatusEstufas[0].inicioReator := '';
	gvl_p.arrStatusEstufas[0].inicioReator := concat(gvl_p.arrStatusEstufas[0].inicioReator,gvl.hora);
	gvl_p.arrStatusEstufas[0].inicioReator := concat(gvl_p.arrStatusEstufas[0].inicioReator,':');
	gvl_p.arrStatusEstufas[0].inicioReator := concat(gvl_p.arrStatusEstufas[0].inicioReator,gvl.minuto);
	gvl_p.arrStatusEstufas[0].inicioReator := concat(gvl_p.arrStatusEstufas[0].inicioReator,' ');
	gvl_p.arrStatusEstufas[0].inicioReator := concat(gvl_p.arrStatusEstufas[0].inicioReator,gvl.dia);
	gvl_p.arrStatusEstufas[0].inicioReator := concat(gvl_p.arrStatusEstufas[0].inicioReator,'/');
	gvl_p.arrStatusEstufas[0].inicioReator := concat(gvl_p.arrStatusEstufas[0].inicioReator,gvl.mes);
	gvl_p.arrStatusEstufas[0].inicioReator := concat(gvl_p.arrStatusEstufas[0].inicioReator,'/');
	gvl_P.arrStatusEstufas[0].inicioReator := concat(gvl_p.arrStatusEstufas[0].inicioReator,gvl.ano);
END_IF

///// DECOMPOR A VARIAVEL FIM DA SECAGEM -----------------------------------------------------------------------------------------------
gvl_p.arrStatusEstufas[0].diaSec := MID(STR:= DT_TO_STRING(gvl_p.arrStatusEstufas[0].fimSecagem) , LEN:= 2, POS:=12);
gvl_p.arrStatusEstufas[0].mesSec := MID(STR:= DT_TO_STRING(gvl_p.arrStatusEstufas[0].fimSecagem), LEN:= 2, POS:=9);
gvl_p.arrStatusEstufas[0].anoSec := MID(STR:= DT_TO_STRING(gvl_p.arrStatusEstufas[0].fimSecagem), LEN:= 2, POS:=6);
gvl_p.arrStatusEstufas[0].horaSec := MID(STR:= DT_TO_STRING(gvl_p.arrStatusEstufas[0].fimSecagem), LEN:= 2, POS:=15);
gvl_p.arrStatusEstufas[0].minutoSec := MID(STR:= DT_TO_STRING(gvl_p.arrStatusEstufas[0].fimSecagem), LEN:= 2, POS:=18);

///// IMPRIMIR A HORA E A DATA DO FIM DA SECAGEM --------------------------------------------------------------------------------------------------------
gvl_p.arrStatusEstufas[0].statusFimSecagem := '';
gvl_p.arrStatusEstufas[0].statusFimSecagem := concat(gvl_p.arrStatusEstufas[0].statusFimSecagem,gvl_p.arrStatusEstufas[0].horaSec);
gvl_p.arrStatusEstufas[0].statusFimSecagem := concat(gvl_p.arrStatusEstufas[0].statusFimSecagem,':');
gvl_p.arrStatusEstufas[0].statusFimSecagem := concat(gvl_p.arrStatusEstufas[0].statusFimSecagem,gvl_p.arrStatusEstufas[0].minutoSec);
gvl_p.arrStatusEstufas[0].statusFimSecagem := concat(gvl_p.arrStatusEstufas[0].statusFimSecagem,' ');
gvl_p.arrStatusEstufas[0].statusFimSecagem := concat(gvl_p.arrStatusEstufas[0].statusFimSecagem,gvl_p.arrStatusEstufas[0].diaSec);
gvl_p.arrStatusEstufas[0].statusFimSecagem := concat(gvl_p.arrStatusEstufas[0].statusFimSecagem,'/');
gvl_p.arrStatusEstufas[0].statusFimSecagem := concat(gvl_p.arrStatusEstufas[0].statusFimSecagem,gvl_p.arrStatusEstufas[0].mesSec);
gvl_p.arrStatusEstufas[0].statusFimSecagem := concat(gvl_p.arrStatusEstufas[0].statusFimSecagem,'/');
gvl_p.arrStatusEstufas[0].statusFimSecagem := concat(gvl_p.arrStatusEstufas[0].statusFimSecagem,gvl_p.arrStatusEstufas[0].anoSec);

///// DECOMPOR A VARIAVEL FIM DA ARMAZENAGEM -------------------------------------------------------------------------------------------
gvl_p.arrStatusEstufas[0].diaArm := MID(STR:= DT_TO_STRING(gvl_p.arrStatusEstufas[0].fimArmazenagem) , LEN:= 2, POS:=12);
gvl_p.arrStatusEstufas[0].mesArm := MID(STR:= DT_TO_STRING(gvl_p.arrStatusEstufas[0].fimArmazenagem), LEN:= 2, POS:=9);
gvl_p.arrStatusEstufas[0].anoArm := MID(STR:= DT_TO_STRING(gvl_P.arrStatusEstufas[0].fimArmazenagem), LEN:= 2, POS:=6);
gvl_p.arrStatusEstufas[0].horaArm := MID(STR:= DT_TO_STRING(gvl_P.arrStatusEstufas[0].fimArmazenagem), LEN:= 2, POS:=15);
gvl_p.arrStatusEstufas[0].minutoArm := MID(STR:= DT_TO_STRING(gvl_p.arrStatusEstufas[0].fimArmazenagem), LEN:= 2, POS:=18);

///// IMPRIMIR A HORA E A DATA DO FIM DA ARMAZENAGEM -----------------------------------------------------------------------------------------------------------
gvl_p.arrStatusEstufas[0].statusFimArmazenagem := '';
gvl_p.arrStatusEstufas[0].statusFimArmazenagem := concat(gvl_p.arrStatusEstufas[0].statusFimArmazenagem,gvl_p.arrStatusEstufas[0].horaArm);
gvl_p.arrStatusEstufas[0].statusFimArmazenagem := concat(gvl_p.arrStatusEstufas[0].statusFimArmazenagem,':');
gvl_p.arrStatusEstufas[0].statusFimArmazenagem := concat(gvl_p.arrStatusEstufas[0].statusFimArmazenagem,gvl_p.arrStatusEstufas[0].minutoArm);
gvl_p.arrStatusEstufas[0].statusFimArmazenagem := concat(gvl_p.arrStatusEstufas[0].statusFimArmazenagem,' ');
gvl_p.arrStatusEstufas[0].statusFimArmazenagem := concat(gvl_p.arrStatusEstufas[0].statusFimArmazenagem,gvl_p.arrStatusEstufas[0].diaArm);
gvl_p.arrStatusEstufas[0].statusFimArmazenagem := concat(gvl_p.arrStatusEstufas[0].statusFimArmazenagem,'/');
gvl_p.arrStatusEstufas[0].statusFimArmazenagem := concat(gvl_p.arrStatusEstufas[0].statusFimArmazenagem,gvl_p.arrStatusEstufas[0].mesArm);
gvl_p.arrStatusEstufas[0].statusFimArmazenagem := concat(gvl_p.arrStatusEstufas[0].statusFimArmazenagem,'/');
gvl_p.arrStatusEstufas[0].statusFimArmazenagem := concat(gvl_p.arrStatusEstufas[0].statusFimArmazenagem,gvl_p.arrStatusEstufas[0].anoArm);

//gvl.permanencia[1]:= DT_TO_TIME(gvl_p.arrStatusEstufas[0].inicioSecagem);
///// GERADOR DE LOG -------------------------------------------------------------

envialog:= 'Secagem Iniciada ESTUFA 019';
gvl.logRegister19:= envialog;

